   1:  PR[GP1:91,1] = PR[GP1:90,1] + 24.010;
   1:  PR[GP1:91,2] = PR[GP1:90,2] + -39.901;
   1:L PR[91] 10mm/sec CNT100;
   1:  PR[GP1:91,1] = PR[GP1:90,1] + 25.299;
   1:  PR[GP1:91,2] = PR[GP1:90,2] + -39.660;
   1:L PR[91] 10mm/sec CNT100;
   1:  PR[GP1:91,1] = PR[GP1:90,1] + 37.312;
   1:  PR[GP1:91,2] = PR[GP1:90,2] + -34.177;
   1:L PR[91] 10mm/sec CNT100;
   1:  PR[GP1:91,1] = PR[GP1:90,1] + 37.829;
   1:  PR[GP1:91,2] = PR[GP1:90,2] + -33.856;
   1:L PR[91] 10mm/sec CNT100;
   1:  PR[GP1:91,1] = PR[GP1:90,1] + 47.713;
   1:  PR[GP1:91,2] = PR[GP1:90,2] + -24.655;
   1:L PR[91] 10mm/sec CNT100;
   1:  PR[GP1:91,1] = PR[GP1:90,1] + 49.263;
   1:  PR[GP1:91,2] = PR[GP1:90,2] + -21.804;
   1:L PR[91] 10mm/sec CNT100;
   1:  PR[GP1:91,1] = PR[GP1:90,1] + 54.196;
   1:  PR[GP1:91,2] = PR[GP1:90,2] + -12.888;
   1:L PR[91] 10mm/sec CNT100;
   1:  PR[GP1:91,1] = PR[GP1:90,1] + 54.207;
   1:  PR[GP1:91,2] = PR[GP1:90,2] + -12.858;
   1:L PR[91] 10mm/sec CNT100;
   1:  PR[GP1:91,1] = PR[GP1:90,1] + 56.443;
   1:  PR[GP1:91,2] = PR[GP1:90,2] + 0.296;
   1:L PR[91] 10mm/sec CNT100;
   1:  PR[GP1:91,1] = PR[GP1:90,1] + 56.432;
   1:  PR[GP1:91,2] = PR[GP1:90,2] + 0.395;
   1:L PR[91] 10mm/sec CNT100;
   1:  PR[GP1:91,1] = PR[GP1:90,1] + 54.197;
   1:  PR[GP1:91,2] = PR[GP1:90,2] + 13.442;
   1:L PR[91] 10mm/sec CNT100;
   1:  PR[GP1:91,1] = PR[GP1:90,1] + 54.186;
   1:  PR[GP1:91,2] = PR[GP1:90,2] + 13.473;
   1:L PR[91] 10mm/sec CNT100;
   1:  PR[GP1:91,1] = PR[GP1:90,1] + 49.263;
   1:  PR[GP1:91,2] = PR[GP1:90,2] + 22.349;
   1:L PR[91] 10mm/sec CNT100;
   1:  PR[GP1:91,1] = PR[GP1:90,1] + 47.678;
   1:  PR[GP1:91,2] = PR[GP1:90,2] + 25.259;
   1:L PR[91] 10mm/sec CNT100;
   1:  PR[GP1:91,1] = PR[GP1:90,1] + 37.759;
   1:  PR[GP1:91,2] = PR[GP1:90,2] + 34.461;
   1:L PR[91] 10mm/sec CNT100;
   1:  PR[GP1:91,1] = PR[GP1:90,1] + 37.238;
   1:  PR[GP1:91,2] = PR[GP1:90,2] + 34.783;
   1:L PR[91] 10mm/sec CNT100;
   1:  PR[GP1:91,1] = PR[GP1:90,1] + 25.194;
   1:  PR[GP1:91,2] = PR[GP1:90,2] + 40.247;
   1:L PR[91] 10mm/sec CNT100;
   1:  PR[GP1:91,1] = PR[GP1:90,1] + 23.898;
   1:  PR[GP1:91,2] = PR[GP1:90,2] + 40.489;
   1:L PR[91] 10mm/sec CNT100;
   1:  PR[GP1:91,1] = PR[GP1:90,1] + 11.139;
   1:  PR[GP1:91,2] = PR[GP1:90,2] + 41.852;
   1:L PR[91] 10mm/sec CNT100;
   1:  PR[GP1:91,1] = PR[GP1:90,1] + 8.485;
   1:  PR[GP1:91,2] = PR[GP1:90,2] + 41.385;
   1:L PR[91] 10mm/sec CNT100;
   1:  PR[GP1:91,1] = PR[GP1:90,1] + -0.260;
   1:  PR[GP1:91,2] = PR[GP1:90,2] + 39.478;
   1:L PR[91] 10mm/sec CNT100;
   1:  PR[GP1:91,1] = PR[GP1:90,1] + -9.009;
   1:  PR[GP1:91,2] = PR[GP1:90,2] + 41.385;
   1:L PR[91] 10mm/sec CNT100;
   1:  PR[GP1:91,1] = PR[GP1:90,1] + -11.665;
   1:  PR[GP1:91,2] = PR[GP1:90,2] + 41.852;
   1:L PR[91] 10mm/sec CNT100;
   1:  PR[GP1:91,1] = PR[GP1:90,1] + -24.425;
   1:  PR[GP1:91,2] = PR[GP1:90,2] + 40.491;
   1:L PR[91] 10mm/sec CNT100;
   1:  PR[GP1:91,1] = PR[GP1:90,1] + -25.720;
   1:  PR[GP1:91,2] = PR[GP1:90,2] + 40.248;
   1:L PR[91] 10mm/sec CNT100;
   1:  PR[GP1:91,1] = PR[GP1:90,1] + -37.764;
   1:  PR[GP1:91,2] = PR[GP1:90,2] + 34.781;
   1:L PR[91] 10mm/sec CNT100;
   1:  PR[GP1:91,1] = PR[GP1:90,1] + -38.285;
   1:  PR[GP1:91,2] = PR[GP1:90,2] + 34.458;
   1:L PR[91] 10mm/sec CNT100;
   1:  PR[GP1:91,1] = PR[GP1:90,1] + -48.204;
   1:  PR[GP1:91,2] = PR[GP1:90,2] + 25.267;
   1:L PR[91] 10mm/sec CNT100;
   1:  PR[GP1:91,1] = PR[GP1:90,1] + -49.790;
   1:  PR[GP1:91,2] = PR[GP1:90,2] + 22.350;
   1:L PR[91] 10mm/sec CNT100;
   1:  PR[GP1:91,1] = PR[GP1:90,1] + -54.712;
   1:  PR[GP1:91,2] = PR[GP1:90,2] + 13.460;
   1:L PR[91] 10mm/sec CNT100;
   1:  PR[GP1:91,1] = PR[GP1:90,1] + -54.724;
   1:  PR[GP1:91,2] = PR[GP1:90,2] + 13.427;
   1:L PR[91] 10mm/sec CNT100;
   1:  PR[GP1:91,1] = PR[GP1:90,1] + -56.969;
   1:  PR[GP1:91,2] = PR[GP1:90,2] + 0.261;
   1:L PR[91] 10mm/sec CNT100;
   1:  PR[GP1:91,1] = PR[GP1:90,1] + -56.959;
   1:  PR[GP1:91,2] = PR[GP1:90,2] + 0.167;
   1:L PR[91] 10mm/sec CNT100;
   1:  PR[GP1:91,1] = PR[GP1:90,1] + -54.734;
   1:  PR[GP1:91,2] = PR[GP1:90,2] + -12.842;
   1:L PR[91] 10mm/sec CNT100;
   1:  PR[GP1:91,1] = PR[GP1:90,1] + -54.722;
   1:  PR[GP1:91,2] = PR[GP1:90,2] + -12.875;
   1:L PR[91] 10mm/sec CNT100;
   1:  PR[GP1:91,1] = PR[GP1:90,1] + -49.791;
   1:  PR[GP1:91,2] = PR[GP1:90,2] + -21.804;
   1:L PR[91] 10mm/sec CNT100;
   1:  PR[GP1:91,1] = PR[GP1:90,1] + -48.225;
   1:  PR[GP1:91,2] = PR[GP1:90,2] + -24.689;
   1:L PR[91] 10mm/sec CNT100;
   1:  PR[GP1:91,1] = PR[GP1:90,1] + -38.356;
   1:  PR[GP1:91,2] = PR[GP1:90,2] + -33.853;
   1:L PR[91] 10mm/sec CNT100;
   1:  PR[GP1:91,1] = PR[GP1:90,1] + -37.838;
   1:  PR[GP1:91,2] = PR[GP1:90,2] + -34.174;
   1:L PR[91] 10mm/sec CNT100;
   1:  PR[GP1:91,1] = PR[GP1:90,1] + -25.826;
   1:  PR[GP1:91,2] = PR[GP1:90,2] + -39.661;
   1:L PR[91] 10mm/sec CNT100;
   1:  PR[GP1:91,1] = PR[GP1:90,1] + -24.537;
   1:  PR[GP1:91,2] = PR[GP1:90,2] + -39.902;
   1:L PR[91] 10mm/sec CNT100;
   1:  PR[GP1:91,1] = PR[GP1:90,1] + -11.796;
   1:  PR[GP1:91,2] = PR[GP1:90,2] + -41.301;
   1:L PR[91] 10mm/sec CNT100;
   1:  PR[GP1:91,1] = PR[GP1:90,1] + -9.923;
   1:  PR[GP1:91,2] = PR[GP1:90,2] + -40.987;
   1:L PR[91] 10mm/sec CNT100;
   1:  PR[GP1:91,1] = PR[GP1:90,1] + -0.262;
   1:  PR[GP1:91,2] = PR[GP1:90,2] + -38.909;
   1:L PR[91] 10mm/sec CNT100;
   1:  PR[GP1:91,1] = PR[GP1:90,1] + 8.960;
   1:  PR[GP1:91,2] = PR[GP1:90,2] + -41.074;
   1:  PR[GP1:91,3] = PR[GP1:90,3] + 91.805;
   1:L PR[91] 10mm/sec CNT100;
   1:  PR[GP1:91,1] = PR[GP1:90,1] + 11.079;
   1:  PR[GP1:91,2] = PR[GP1:90,2] + -41.430;
   1:L PR[91] 10mm/sec CNT100;
   1:  PR[GP1:91,1] = PR[GP1:90,1] + 23.609;
   1:  PR[GP1:91,2] = PR[GP1:90,2] + -40.053;
   1:L PR[91] 10mm/sec CNT100;
   1:  PR[GP1:91,1] = PR[GP1:90,1] + 25.173;
   1:  PR[GP1:91,2] = PR[GP1:90,2] + -39.761;
   1:L PR[91] 10mm/sec CNT100;
   1:  PR[GP1:91,1] = PR[GP1:90,1] + 36.986;
   1:  PR[GP1:91,2] = PR[GP1:90,2] + -34.368;
   1:L PR[91] 10mm/sec CNT100;
   1:  PR[GP1:91,1] = PR[GP1:90,1] + 37.751;
   1:  PR[GP1:91,2] = PR[GP1:90,2] + -33.894;
   1:L PR[91] 10mm/sec CNT100;
   1:  PR[GP1:91,1] = PR[GP1:90,1] + 47.467;
   1:  PR[GP1:91,2] = PR[GP1:90,2] + -24.863;
   1:L PR[91] 10mm/sec CNT100;
   1:  PR[GP1:91,1] = PR[GP1:90,1] + 47.597;
   1:  PR[GP1:91,2] = PR[GP1:90,2] + -24.706;
   1:L PR[91] 10mm/sec CNT100;
   1:  PR[GP1:91,1] = PR[GP1:90,1] + 54.014;
   1:  PR[GP1:91,2] = PR[GP1:90,2] + -12.903;
   1:L PR[91] 10mm/sec CNT100;
   1:  PR[GP1:91,1] = PR[GP1:90,1] + 56.264;
   1:  PR[GP1:91,2] = PR[GP1:90,2] + 0.291;
   1:L PR[91] 10mm/sec CNT100;
   1:  PR[GP1:91,1] = PR[GP1:90,1] + 54.005;
   1:  PR[GP1:91,2] = PR[GP1:90,2] + 13.485;
   1:L PR[91] 10mm/sec CNT100;
   1:  PR[GP1:91,1] = PR[GP1:90,1] + 47.562;
   1:  PR[GP1:91,2] = PR[GP1:90,2] + 25.309;
   1:L PR[91] 10mm/sec CNT100;
   1:  PR[GP1:91,1] = PR[GP1:90,1] + 47.431;
   1:  PR[GP1:91,2] = PR[GP1:90,2] + 25.467;
   1:L PR[91] 10mm/sec CNT100;
   1:  PR[GP1:91,1] = PR[GP1:90,1] + 37.682;
   1:  PR[GP1:91,2] = PR[GP1:90,2] + 34.498;
   1:L PR[91] 10mm/sec CNT100;
   1:  PR[GP1:91,1] = PR[GP1:90,1] + 36.914;
   1:  PR[GP1:91,2] = PR[GP1:90,2] + 34.974;
   1:L PR[91] 10mm/sec CNT100;
   1:  PR[GP1:91,1] = PR[GP1:90,1] + 25.069;
   1:  PR[GP1:91,2] = PR[GP1:90,2] + 40.347;
   1:L PR[91] 10mm/sec CNT100;
   1:  PR[GP1:91,1] = PR[GP1:90,1] + 23.500;
   1:  PR[GP1:91,2] = PR[GP1:90,2] + 40.641;
   1:L PR[91] 10mm/sec CNT100;
   1:  PR[GP1:91,1] = PR[GP1:90,1] + 10.952;
   1:  PR[GP1:91,2] = PR[GP1:90,2] + 41.981;
   1:L PR[91] 10mm/sec CNT100;
   1:  PR[GP1:91,1] = PR[GP1:90,1] + 7.952;
   1:  PR[GP1:91,2] = PR[GP1:90,2] + 41.453;
   1:L PR[91] 10mm/sec CNT100;
   1:  PR[GP1:91,1] = PR[GP1:90,1] + -0.260;
   1:  PR[GP1:91,2] = PR[GP1:90,2] + 39.662;
   1:L PR[91] 10mm/sec CNT100;
   1:  PR[GP1:91,1] = PR[GP1:90,1] + -8.475;
   1:  PR[GP1:91,2] = PR[GP1:90,2] + 41.453;
   1:L PR[91] 10mm/sec CNT100;
   1:  PR[GP1:91,1] = PR[GP1:90,1] + -11.478;
   1:  PR[GP1:91,2] = PR[GP1:90,2] + 41.980;
   1:L PR[91] 10mm/sec CNT100;
   1:  PR[GP1:91,1] = PR[GP1:90,1] + -24.026;
   1:  PR[GP1:91,2] = PR[GP1:90,2] + 40.642;
   1:L PR[91] 10mm/sec CNT100;
   1:  PR[GP1:91,1] = PR[GP1:90,1] + -25.595;
   1:  PR[GP1:91,2] = PR[GP1:90,2] + 40.348;
   1:L PR[91] 10mm/sec CNT100;
   1:  PR[GP1:91,1] = PR[GP1:90,1] + -37.440;
   1:  PR[GP1:91,2] = PR[GP1:90,2] + 34.971;
   1:L PR[91] 10mm/sec CNT100;
   1:  PR[GP1:91,1] = PR[GP1:90,1] + -38.208;
   1:  PR[GP1:91,2] = PR[GP1:90,2] + 34.496;
   1:L PR[91] 10mm/sec CNT100;
   1:  PR[GP1:91,1] = PR[GP1:90,1] + -47.957;
   1:  PR[GP1:91,2] = PR[GP1:90,2] + 25.475;
   1:L PR[91] 10mm/sec CNT100;
   1:  PR[GP1:91,1] = PR[GP1:90,1] + -48.088;
   1:  PR[GP1:91,2] = PR[GP1:90,2] + 25.317;
   1:L PR[91] 10mm/sec CNT100;
   1:  PR[GP1:91,1] = PR[GP1:90,1] + -54.531;
   1:  PR[GP1:91,2] = PR[GP1:90,2] + 13.474;
   1:L PR[91] 10mm/sec CNT100;
   1:  PR[GP1:91,1] = PR[GP1:90,1] + -56.791;
   1:  PR[GP1:91,2] = PR[GP1:90,2] + 0.267;
   1:L PR[91] 10mm/sec CNT100;
   1:  PR[GP1:91,1] = PR[GP1:90,1] + -54.541;
   1:  PR[GP1:91,2] = PR[GP1:90,2] + -12.886;
   1:L PR[91] 10mm/sec CNT100;
   1:  PR[GP1:91,1] = PR[GP1:90,1] + -48.123;
   1:  PR[GP1:91,2] = PR[GP1:90,2] + -24.714;
   1:L PR[91] 10mm/sec CNT100;
   1:  PR[GP1:91,1] = PR[GP1:90,1] + -47.994;
   1:  PR[GP1:91,2] = PR[GP1:90,2] + -24.870;
   1:L PR[91] 10mm/sec CNT100;
   1:  PR[GP1:91,1] = PR[GP1:90,1] + -38.278;
   1:  PR[GP1:91,2] = PR[GP1:90,2] + -33.892;
   1:L PR[91] 10mm/sec CNT100;
   1:  PR[GP1:91,1] = PR[GP1:90,1] + -37.513;
   1:  PR[GP1:91,2] = PR[GP1:90,2] + -34.365;
   1:L PR[91] 10mm/sec CNT100;
   1:  PR[GP1:91,1] = PR[GP1:90,1] + -25.700;
   1:  PR[GP1:91,2] = PR[GP1:90,2] + -39.762;
   1:L PR[91] 10mm/sec CNT100;
   1:  PR[GP1:91,1] = PR[GP1:90,1] + -24.136;
   1:  PR[GP1:91,2] = PR[GP1:90,2] + -40.054;
   1:L PR[91] 10mm/sec CNT100;
   1:  PR[GP1:91,1] = PR[GP1:90,1] + -11.606;
   1:  PR[GP1:91,2] = PR[GP1:90,2] + -41.429;
   1:L PR[91] 10mm/sec CNT100;
   1:  PR[GP1:91,1] = PR[GP1:90,1] + -9.485;
   1:  PR[GP1:91,2] = PR[GP1:90,2] + -41.074;
   1:L PR[91] 10mm/sec CNT100;
   1:  PR[GP1:91,1] = PR[GP1:90,1] + -0.262;
   1:  PR[GP1:91,2] = PR[GP1:90,2] + -39.090;
   1:L PR[91] 10mm/sec CNT100;
   1:  PR[GP1:91,1] = PR[GP1:90,1] + 8.523;
   1:  PR[GP1:91,2] = PR[GP1:90,2] + -41.161;
   1:  PR[GP1:91,3] = PR[GP1:90,3] + 92.415;
   1:L PR[91] 10mm/sec CNT100;
   1:  PR[GP1:91,1] = PR[GP1:90,1] + 10.890;
   1:  PR[GP1:91,2] = PR[GP1:90,2] + -41.558;
   1:L PR[91] 10mm/sec CNT100;
   1:  PR[GP1:91,1] = PR[GP1:90,1] + 23.209;
   1:  PR[GP1:91,2] = PR[GP1:90,2] + -40.205;
   1:L PR[91] 10mm/sec CNT100;
   1:  PR[GP1:91,1] = PR[GP1:90,1] + 25.047;
   1:  PR[GP1:91,2] = PR[GP1:90,2] + -39.861;
   1:L PR[91] 10mm/sec CNT100;
   1:  PR[GP1:91,1] = PR[GP1:90,1] + 36.661;
   1:  PR[GP1:91,2] = PR[GP1:90,2] + -34.559;
   1:L PR[91] 10mm/sec CNT100;
   1:  PR[GP1:91,1] = PR[GP1:90,1] + 37.673;
   1:  PR[GP1:91,2] = PR[GP1:90,2] + -33.933;
   1:L PR[91] 10mm/sec CNT100;
   1:  PR[GP1:91,1] = PR[GP1:90,1] + 47.225;
   1:  PR[GP1:91,2] = PR[GP1:90,2] + -25.053;
   1:L PR[91] 10mm/sec CNT100;
   1:  PR[GP1:91,1] = PR[GP1:90,1] + 47.499;
   1:  PR[GP1:91,2] = PR[GP1:90,2] + -24.723;
   1:L PR[91] 10mm/sec CNT100;
   1:  PR[GP1:91,1] = PR[GP1:90,1] + 53.845;
   1:  PR[GP1:91,2] = PR[GP1:90,2] + -13.048;
   1:L PR[91] 10mm/sec CNT100;
   1:  PR[GP1:91,1] = PR[GP1:90,1] + 53.896;
   1:  PR[GP1:91,2] = PR[GP1:90,2] + -12.932;
   1:L PR[91] 10mm/sec CNT100;
   1:  PR[GP1:91,1] = PR[GP1:90,1] + 56.107;
   1:  PR[GP1:91,2] = PR[GP1:90,2] + 0.224;
   1:L PR[91] 10mm/sec CNT100;
   1:  PR[GP1:91,2] = PR[GP1:90,2] + 0.232;
   1:L PR[91] 10mm/sec CNT100;
   1:  PR[GP1:91,1] = PR[GP1:90,1] + 54.998;
   1:  PR[GP1:91,2] = PR[GP1:90,2] + 6.763;
   1:L PR[91] 10mm/sec CNT100;
   1:  PR[GP1:91,1] = PR[GP1:90,1] + 53.886;
   1:  PR[GP1:91,2] = PR[GP1:90,2] + 13.518;
   1:L PR[91] 10mm/sec CNT100;
   1:  PR[GP1:91,1] = PR[GP1:90,1] + 53.835;
   1:  PR[GP1:91,2] = PR[GP1:90,2] + 13.633;
   1:L PR[91] 10mm/sec CNT100;
   1:  PR[GP1:91,1] = PR[GP1:90,1] + 47.465;
   1:  PR[GP1:91,2] = PR[GP1:90,2] + 25.325;
   1:L PR[91] 10mm/sec CNT100;
   1:  PR[GP1:91,1] = PR[GP1:90,1] + 47.190;
   1:  PR[GP1:91,2] = PR[GP1:90,2] + 25.657;
   1:L PR[91] 10mm/sec CNT100;
   1:  PR[GP1:91,1] = PR[GP1:90,1] + 37.605;
   1:  PR[GP1:91,2] = PR[GP1:90,2] + 34.536;
   1:L PR[91] 10mm/sec CNT100;
   1:  PR[GP1:91,1] = PR[GP1:90,1] + 36.590;
   1:  PR[GP1:91,2] = PR[GP1:90,2] + 35.164;
   1:L PR[91] 10mm/sec CNT100;
   1:  PR[GP1:91,1] = PR[GP1:90,1] + 24.945;
   1:  PR[GP1:91,2] = PR[GP1:90,2] + 40.447;
   1:L PR[91] 10mm/sec CNT100;
   1:  PR[GP1:91,1] = PR[GP1:90,1] + 23.101;
   1:  PR[GP1:91,2] = PR[GP1:90,2] + 40.792;
   1:L PR[91] 10mm/sec CNT100;
   1:  PR[GP1:91,1] = PR[GP1:90,1] + 10.765;
   1:  PR[GP1:91,2] = PR[GP1:90,2] + 42.109;
   1:L PR[91] 10mm/sec CNT100;
   1:  PR[GP1:91,1] = PR[GP1:90,1] + 7.418;
   1:  PR[GP1:91,2] = PR[GP1:90,2] + 41.521;
   1:L PR[91] 10mm/sec CNT100;
   1:  PR[GP1:91,1] = PR[GP1:90,1] + -0.260;
   1:  PR[GP1:91,2] = PR[GP1:90,2] + 39.846;
   1:L PR[91] 10mm/sec CNT100;
   1:  PR[GP1:91,1] = PR[GP1:90,1] + -7.941;
   1:  PR[GP1:91,2] = PR[GP1:90,2] + 41.520;
   1:L PR[91] 10mm/sec CNT100;
   1:  PR[GP1:91,1] = PR[GP1:90,1] + -11.291;
   1:  PR[GP1:91,2] = PR[GP1:90,2] + 42.109;
   1:L PR[91] 10mm/sec CNT100;
   1:  PR[GP1:91,1] = PR[GP1:90,1] + -23.628;
   1:  PR[GP1:91,2] = PR[GP1:90,2] + 40.793;
   1:L PR[91] 10mm/sec CNT100;
   1:  PR[GP1:91,1] = PR[GP1:90,1] + -25.471;
   1:  PR[GP1:91,2] = PR[GP1:90,2] + 40.448;
   1:L PR[91] 10mm/sec CNT100;
   1:  PR[GP1:91,1] = PR[GP1:90,1] + -37.116;
   1:  PR[GP1:91,2] = PR[GP1:90,2] + 35.162;
   1:L PR[91] 10mm/sec CNT100;
   1:  PR[GP1:91,1] = PR[GP1:90,1] + -38.131;
   1:  PR[GP1:91,2] = PR[GP1:90,2] + 34.533;
   1:L PR[91] 10mm/sec CNT100;
   1:  PR[GP1:91,1] = PR[GP1:90,1] + -47.716;
   1:  PR[GP1:91,2] = PR[GP1:90,2] + 25.664;
   1:L PR[91] 10mm/sec CNT100;
   1:  PR[GP1:91,1] = PR[GP1:90,1] + -47.991;
   1:  PR[GP1:91,2] = PR[GP1:90,2] + 25.333;
   1:L PR[91] 10mm/sec CNT100;
   1:  PR[GP1:91,1] = PR[GP1:90,1] + -54.361;
   1:  PR[GP1:91,2] = PR[GP1:90,2] + 13.620;
   1:L PR[91] 10mm/sec CNT100;
   1:  PR[GP1:91,1] = PR[GP1:90,1] + -54.413;
   1:  PR[GP1:91,2] = PR[GP1:90,2] + 13.503;
   1:L PR[91] 10mm/sec CNT100;
   1:  PR[GP1:91,1] = PR[GP1:90,1] + -56.633;
   1:  PR[GP1:91,2] = PR[GP1:90,2] + 0.334;
   1:L PR[91] 10mm/sec CNT100;
   1:  PR[GP1:91,2] = PR[GP1:90,2] + 0.326;
   1:L PR[91] 10mm/sec CNT100;
   1:  PR[GP1:91,1] = PR[GP1:90,1] + -55.528;
   1:  PR[GP1:91,2] = PR[GP1:90,2] + -6.190;
   1:L PR[91] 10mm/sec CNT100;
   1:  PR[GP1:91,1] = PR[GP1:90,1] + -54.439;
   1:  PR[GP1:91,2] = PR[GP1:90,2] + -12.777;
   1:L PR[91] 10mm/sec CNT100;
   1:  PR[GP1:91,1] = PR[GP1:90,1] + -54.419;
   1:  PR[GP1:91,2] = PR[GP1:90,2] + -12.926;
   1:L PR[91] 10mm/sec CNT100;
   1:  PR[GP1:91,1] = PR[GP1:90,1] + -54.371;
   1:  PR[GP1:91,2] = PR[GP1:90,2] + -13.034;
   1:L PR[91] 10mm/sec CNT100;
   1:  PR[GP1:91,1] = PR[GP1:90,1] + -48.026;
   1:  PR[GP1:91,2] = PR[GP1:90,2] + -24.730;
   1:L PR[91] 10mm/sec CNT100;
   1:  PR[GP1:91,1] = PR[GP1:90,1] + -47.752;
   1:  PR[GP1:91,2] = PR[GP1:90,2] + -25.060;
   1:L PR[91] 10mm/sec CNT100;
   1:  PR[GP1:91,1] = PR[GP1:90,1] + -38.199;
   1:  PR[GP1:91,2] = PR[GP1:90,2] + -33.930;
   1:L PR[91] 10mm/sec CNT100;
   1:  PR[GP1:91,1] = PR[GP1:90,1] + -37.188;
   1:  PR[GP1:91,2] = PR[GP1:90,2] + -34.557;
   1:L PR[91] 10mm/sec CNT100;
   1:  PR[GP1:91,1] = PR[GP1:90,1] + -25.573;
   1:  PR[GP1:91,2] = PR[GP1:90,2] + -39.862;
   1:L PR[91] 10mm/sec CNT100;
   1:  PR[GP1:91,1] = PR[GP1:90,1] + -23.736;
   1:  PR[GP1:91,2] = PR[GP1:90,2] + -40.206;
   1:L PR[91] 10mm/sec CNT100;
   1:  PR[GP1:91,1] = PR[GP1:90,1] + -11.417;
   1:  PR[GP1:91,2] = PR[GP1:90,2] + -41.558;
   1:L PR[91] 10mm/sec CNT100;
   1:  PR[GP1:91,1] = PR[GP1:90,1] + -9.047;
   1:  PR[GP1:91,2] = PR[GP1:90,2] + -41.160;
   1:L PR[91] 10mm/sec CNT100;
   1:  PR[GP1:91,1] = PR[GP1:90,1] + -0.262;
   1:  PR[GP1:91,2] = PR[GP1:90,2] + -39.271;
   1:L PR[91] 10mm/sec CNT100;
   1:  PR[GP1:91,1] = PR[GP1:90,1] + 8.085;
   1:  PR[GP1:91,2] = PR[GP1:90,2] + -41.247;
   1:  PR[GP1:91,3] = PR[GP1:90,3] + 93.025;
   1:L PR[91] 10mm/sec CNT100;
   1:  PR[GP1:91,1] = PR[GP1:90,1] + 10.700;
   1:  PR[GP1:91,2] = PR[GP1:90,2] + -41.687;
   1:L PR[91] 10mm/sec CNT100;
   1:  PR[GP1:91,1] = PR[GP1:90,1] + 22.808;
   1:  PR[GP1:91,2] = PR[GP1:90,2] + -40.356;
   1:L PR[91] 10mm/sec CNT100;
   1:  PR[GP1:91,1] = PR[GP1:90,1] + 24.920;
   1:  PR[GP1:91,2] = PR[GP1:90,2] + -39.962;
   1:L PR[91] 10mm/sec CNT100;
   1:  PR[GP1:91,1] = PR[GP1:90,1] + 36.336;
   1:  PR[GP1:91,2] = PR[GP1:90,2] + -34.751;
   1:L PR[91] 10mm/sec CNT100;
   1:  PR[GP1:91,1] = PR[GP1:90,1] + 37.594;
   1:  PR[GP1:91,2] = PR[GP1:90,2] + -33.971;
   1:L PR[91] 10mm/sec CNT100;
   1:  PR[GP1:91,1] = PR[GP1:90,1] + 46.983;
   1:  PR[GP1:91,2] = PR[GP1:90,2] + -25.243;
   1:L PR[91] 10mm/sec CNT100;
   1:  PR[GP1:91,1] = PR[GP1:90,1] + 47.402;
   1:  PR[GP1:91,2] = PR[GP1:90,2] + -24.739;
   1:L PR[91] 10mm/sec CNT100;
   1:  PR[GP1:91,1] = PR[GP1:90,1] + 53.638;
   1:  PR[GP1:91,2] = PR[GP1:90,2] + -13.265;
   1:L PR[91] 10mm/sec CNT100;
   1:  PR[GP1:91,1] = PR[GP1:90,1] + 53.783;
   1:  PR[GP1:91,2] = PR[GP1:90,2] + -12.937;
   1:L PR[91] 10mm/sec CNT100;
   1:  PR[GP1:91,1] = PR[GP1:90,1] + 55.956;
   1:  PR[GP1:91,2] = PR[GP1:90,2] + -0.005;
   1:L PR[91] 10mm/sec CNT100;
   1:  PR[GP1:91,1] = PR[GP1:90,1] + 55.960;
   1:  PR[GP1:91,2] = PR[GP1:90,2] + 0.234;
   1:L PR[91] 10mm/sec CNT100;
   1:  PR[GP1:91,1] = PR[GP1:90,1] + 53.823;
   1:  PR[GP1:91,2] = PR[GP1:90,2] + 13.152;
   1:L PR[91] 10mm/sec CNT100;
   1:  PR[GP1:91,1] = PR[GP1:90,1] + 53.770;
   1:  PR[GP1:91,2] = PR[GP1:90,2] + 13.530;
   1:L PR[91] 10mm/sec CNT100;
   1:  PR[GP1:91,1] = PR[GP1:90,1] + 53.629;
   1:  PR[GP1:91,2] = PR[GP1:90,2] + 13.849;
   1:L PR[91] 10mm/sec CNT100;
   1:  PR[GP1:91,1] = PR[GP1:90,1] + 47.368;
   1:  PR[GP1:91,2] = PR[GP1:90,2] + 25.341;
   1:L PR[91] 10mm/sec CNT100;
   1:  PR[GP1:91,1] = PR[GP1:90,1] + 46.948;
   1:  PR[GP1:91,2] = PR[GP1:90,2] + 25.846;
   1:L PR[91] 10mm/sec CNT100;
   1:  PR[GP1:91,1] = PR[GP1:90,1] + 37.528;
   1:  PR[GP1:91,2] = PR[GP1:90,2] + 34.573;
   1:L PR[91] 10mm/sec CNT100;
   1:  PR[GP1:91,1] = PR[GP1:90,1] + 36.265;
   1:  PR[GP1:91,2] = PR[GP1:90,2] + 35.355;
   1:L PR[91] 10mm/sec CNT100;
   1:  PR[GP1:91,1] = PR[GP1:90,1] + 24.820;
   1:  PR[GP1:91,2] = PR[GP1:90,2] + 40.547;
   1:L PR[91] 10mm/sec CNT100;
   1:  PR[GP1:91,1] = PR[GP1:90,1] + 22.702;
   1:  PR[GP1:91,2] = PR[GP1:90,2] + 40.943;
   1:L PR[91] 10mm/sec CNT100;
   1:  PR[GP1:91,1] = PR[GP1:90,1] + 10.577;
   1:  PR[GP1:91,2] = PR[GP1:90,2] + 42.238;
   1:L PR[91] 10mm/sec CNT100;
   1:  PR[GP1:91,1] = PR[GP1:90,1] + 6.885;
   1:  PR[GP1:91,2] = PR[GP1:90,2] + 41.588;
   1:L PR[91] 10mm/sec CNT100;
   1:  PR[GP1:91,1] = PR[GP1:90,1] + -0.260;
   1:  PR[GP1:91,2] = PR[GP1:90,2] + 40.030;
   1:L PR[91] 10mm/sec CNT100;
   1:  PR[GP1:91,1] = PR[GP1:90,1] + -7.407;
   1:  PR[GP1:91,2] = PR[GP1:90,2] + 41.588;
   1:L PR[91] 10mm/sec CNT100;
   1:  PR[GP1:91,1] = PR[GP1:90,1] + -11.104;
   1:  PR[GP1:91,2] = PR[GP1:90,2] + 42.237;
   1:L PR[91] 10mm/sec CNT100;
   1:  PR[GP1:91,1] = PR[GP1:90,1] + -23.229;
   1:  PR[GP1:91,2] = PR[GP1:90,2] + 40.944;
   1:L PR[91] 10mm/sec CNT100;
   1:  PR[GP1:91,1] = PR[GP1:90,1] + -25.346;
   1:  PR[GP1:91,2] = PR[GP1:90,2] + 40.548;
   1:L PR[91] 10mm/sec CNT100;
   1:  PR[GP1:91,1] = PR[GP1:90,1] + -36.792;
   1:  PR[GP1:91,2] = PR[GP1:90,2] + 35.352;
   1:L PR[91] 10mm/sec CNT100;
   1:  PR[GP1:91,1] = PR[GP1:90,1] + -38.054;
   1:  PR[GP1:91,2] = PR[GP1:90,2] + 34.571;
   1:L PR[91] 10mm/sec CNT100;
   1:  PR[GP1:91,1] = PR[GP1:90,1] + -47.475;
   1:  PR[GP1:91,2] = PR[GP1:90,2] + 25.854;
   1:L PR[91] 10mm/sec CNT100;
   1:  PR[GP1:91,1] = PR[GP1:90,1] + -47.894;
   1:  PR[GP1:91,2] = PR[GP1:90,2] + 25.349;
   1:L PR[91] 10mm/sec CNT100;
   1:  PR[GP1:91,1] = PR[GP1:90,1] + -54.155;
   1:  PR[GP1:91,2] = PR[GP1:90,2] + 13.836;
   1:L PR[91] 10mm/sec CNT100;
   1:  PR[GP1:91,1] = PR[GP1:90,1] + -54.300;
   1:  PR[GP1:91,2] = PR[GP1:90,2] + 13.508;
   1:L PR[91] 10mm/sec CNT100;
   1:  PR[GP1:91,1] = PR[GP1:90,1] + -56.482;
   1:  PR[GP1:91,2] = PR[GP1:90,2] + 0.565;
   1:L PR[91] 10mm/sec CNT100;
   1:  PR[GP1:91,1] = PR[GP1:90,1] + -56.485;
   1:  PR[GP1:91,2] = PR[GP1:90,2] + 0.316;
   1:L PR[91] 10mm/sec CNT100;
   1:  PR[GP1:91,1] = PR[GP1:90,1] + -54.358;
   1:  PR[GP1:91,2] = PR[GP1:90,2] + -12.554;
   1:L PR[91] 10mm/sec CNT100;
   1:  PR[GP1:91,1] = PR[GP1:90,1] + -54.306;
   1:  PR[GP1:91,2] = PR[GP1:90,2] + -12.931;
   1:L PR[91] 10mm/sec CNT100;
   1:  PR[GP1:91,1] = PR[GP1:90,1] + -54.165;
   1:  PR[GP1:91,2] = PR[GP1:90,2] + -13.251;
   1:L PR[91] 10mm/sec CNT100;
   1:  PR[GP1:91,1] = PR[GP1:90,1] + -47.928;
   1:  PR[GP1:91,2] = PR[GP1:90,2] + -24.747;
   1:L PR[91] 10mm/sec CNT100;
   1:  PR[GP1:91,1] = PR[GP1:90,1] + -47.510;
   1:  PR[GP1:91,2] = PR[GP1:90,2] + -25.251;
   1:L PR[91] 10mm/sec CNT100;
   1:  PR[GP1:91,1] = PR[GP1:90,1] + -38.121;
   1:  PR[GP1:91,2] = PR[GP1:90,2] + -33.968;
   1:L PR[91] 10mm/sec CNT100;
   1:  PR[GP1:91,1] = PR[GP1:90,1] + -36.862;
   1:  PR[GP1:91,2] = PR[GP1:90,2] + -34.748;
   1:L PR[91] 10mm/sec CNT100;
   1:  PR[GP1:91,1] = PR[GP1:90,1] + -25.447;
   1:  PR[GP1:91,2] = PR[GP1:90,2] + -39.962;
   1:L PR[91] 10mm/sec CNT100;
   1:  PR[GP1:91,1] = PR[GP1:90,1] + -23.336;
   1:  PR[GP1:91,2] = PR[GP1:90,2] + -40.357;
   1:L PR[91] 10mm/sec CNT100;
   1:  PR[GP1:91,1] = PR[GP1:90,1] + -11.228;
   1:  PR[GP1:91,2] = PR[GP1:90,2] + -41.686;
   1:L PR[91] 10mm/sec CNT100;
   1:  PR[GP1:91,1] = PR[GP1:90,1] + -8.609;
   1:  PR[GP1:91,2] = PR[GP1:90,2] + -41.247;
   1:L PR[91] 10mm/sec CNT100;
   1:  PR[GP1:91,1] = PR[GP1:90,1] + -0.262;
   1:  PR[GP1:91,2] = PR[GP1:90,2] + -39.452;
   1:L PR[91] 10mm/sec CNT100;
   1:  PR[GP1:91,1] = PR[GP1:90,1] + 7.647;
   1:  PR[GP1:91,2] = PR[GP1:90,2] + -41.334;
   1:  PR[GP1:91,3] = PR[GP1:90,3] + 93.635;
   1:L PR[91] 10mm/sec CNT100;
   1:  PR[GP1:91,1] = PR[GP1:90,1] + 10.511;
   1:  PR[GP1:91,2] = PR[GP1:90,2] + -41.815;
   1:L PR[91] 10mm/sec CNT100;
   1:  PR[GP1:91,1] = PR[GP1:90,1] + 22.408;
   1:  PR[GP1:91,2] = PR[GP1:90,2] + -40.508;
   1:L PR[91] 10mm/sec CNT100;
   1:  PR[GP1:91,1] = PR[GP1:90,1] + 24.794;
   1:  PR[GP1:91,2] = PR[GP1:90,2] + -40.062;
   1:L PR[91] 10mm/sec CNT100;
   1:  PR[GP1:91,1] = PR[GP1:90,1] + 36.010;
   1:  PR[GP1:91,2] = PR[GP1:90,2] + -34.942;
   1:L PR[91] 10mm/sec CNT100;
   1:  PR[GP1:91,1] = PR[GP1:90,1] + 37.516;
   1:  PR[GP1:91,2] = PR[GP1:90,2] + -34.009;
   1:L PR[91] 10mm/sec CNT100;
   1:  PR[GP1:91,1] = PR[GP1:90,1] + 46.741;
   1:  PR[GP1:91,2] = PR[GP1:90,2] + -25.434;
   1:L PR[91] 10mm/sec CNT100;
   1:  PR[GP1:91,1] = PR[GP1:90,1] + 47.304;
   1:  PR[GP1:91,2] = PR[GP1:90,2] + -24.756;
   1:L PR[91] 10mm/sec CNT100;
   1:  PR[GP1:91,1] = PR[GP1:90,1] + 53.432;
   1:  PR[GP1:91,2] = PR[GP1:90,2] + -13.481;
   1:L PR[91] 10mm/sec CNT100;
   1:  PR[GP1:91,1] = PR[GP1:90,1] + 53.670;
   1:  PR[GP1:91,2] = PR[GP1:90,2] + -12.943;
   1:L PR[91] 10mm/sec CNT100;
   1:  PR[GP1:91,1] = PR[GP1:90,1] + 55.805;
   1:  PR[GP1:91,2] = PR[GP1:90,2] + -0.237;
   1:L PR[91] 10mm/sec CNT100;
   1:  PR[GP1:91,1] = PR[GP1:90,1] + 55.809;
   1:  PR[GP1:91,2] = PR[GP1:90,2] + 0.075;
   1:L PR[91] 10mm/sec CNT100;
   1:  PR[GP1:91,1] = PR[GP1:90,1] + 55.836;
   1:  PR[GP1:91,2] = PR[GP1:90,2] + 0.271;
   1:L PR[91] 10mm/sec CNT100;
   1:  PR[GP1:91,1] = PR[GP1:90,1] + 53.742;
   1:  PR[GP1:91,2] = PR[GP1:90,2] + 12.928;
   1:L PR[91] 10mm/sec CNT100;
   1:  PR[GP1:91,1] = PR[GP1:90,1] + 53.657;
   1:  PR[GP1:91,2] = PR[GP1:90,2] + 13.534;
   1:L PR[91] 10mm/sec CNT100;
   1:  PR[GP1:91,1] = PR[GP1:90,1] + 53.423;
   1:  PR[GP1:91,2] = PR[GP1:90,2] + 14.065;
   1:L PR[91] 10mm/sec CNT100;
   1:  PR[GP1:91,1] = PR[GP1:90,1] + 47.271;
   1:  PR[GP1:91,2] = PR[GP1:90,2] + 25.357;
   1:L PR[91] 10mm/sec CNT100;
   1:  PR[GP1:91,1] = PR[GP1:90,1] + 46.707;
   1:  PR[GP1:91,2] = PR[GP1:90,2] + 26.036;
   1:L PR[91] 10mm/sec CNT100;
   1:  PR[GP1:91,1] = PR[GP1:90,1] + 37.450;
   1:  PR[GP1:91,2] = PR[GP1:90,2] + 34.611;
   1:L PR[91] 10mm/sec CNT100;
   1:  PR[GP1:91,1] = PR[GP1:90,1] + 35.941;
   1:  PR[GP1:91,2] = PR[GP1:90,2] + 35.545;
   1:L PR[91] 10mm/sec CNT100;
   1:  PR[GP1:91,1] = PR[GP1:90,1] + 24.696;
   1:  PR[GP1:91,2] = PR[GP1:90,2] + 40.647;
   1:L PR[91] 10mm/sec CNT100;
   1:  PR[GP1:91,1] = PR[GP1:90,1] + 22.304;
   1:  PR[GP1:91,2] = PR[GP1:90,2] + 41.094;
   1:L PR[91] 10mm/sec CNT100;
   1:  PR[GP1:91,1] = PR[GP1:90,1] + 10.390;
   1:  PR[GP1:91,2] = PR[GP1:90,2] + 42.366;
   1:L PR[91] 10mm/sec CNT100;
   1:  PR[GP1:91,1] = PR[GP1:90,1] + 6.351;
   1:  PR[GP1:91,2] = PR[GP1:90,2] + 41.656;
   1:L PR[91] 10mm/sec CNT100;
   1:  PR[GP1:91,1] = PR[GP1:90,1] + -0.260;
   1:  PR[GP1:91,2] = PR[GP1:90,2] + 40.214;
   1:L PR[91] 10mm/sec CNT100;
   1:  PR[GP1:91,1] = PR[GP1:90,1] + -6.874;
   1:  PR[GP1:91,2] = PR[GP1:90,2] + 41.656;
   1:L PR[91] 10mm/sec CNT100;
   1:  PR[GP1:91,1] = PR[GP1:90,1] + -10.917;
   1:  PR[GP1:91,2] = PR[GP1:90,2] + 42.366;
   1:L PR[91] 10mm/sec CNT100;
   1:  PR[GP1:91,1] = PR[GP1:90,1] + -22.831;
   1:  PR[GP1:91,2] = PR[GP1:90,2] + 41.095;
   1:L PR[91] 10mm/sec CNT100;
   1:  PR[GP1:91,1] = PR[GP1:90,1] + -25.222;
   1:  PR[GP1:91,2] = PR[GP1:90,2] + 40.648;
   1:L PR[91] 10mm/sec CNT100;
   1:  PR[GP1:91,1] = PR[GP1:90,1] + -36.468;
   1:  PR[GP1:91,2] = PR[GP1:90,2] + 35.543;
   1:L PR[91] 10mm/sec CNT100;
   1:  PR[GP1:91,1] = PR[GP1:90,1] + -37.976;
   1:  PR[GP1:91,2] = PR[GP1:90,2] + 34.608;
   1:L PR[91] 10mm/sec CNT100;
   1:  PR[GP1:91,1] = PR[GP1:90,1] + -47.233;
   1:  PR[GP1:91,2] = PR[GP1:90,2] + 26.043;
   1:L PR[91] 10mm/sec CNT100;
   1:  PR[GP1:91,1] = PR[GP1:90,1] + -47.797;
   1:  PR[GP1:91,2] = PR[GP1:90,2] + 25.365;
   1:L PR[91] 10mm/sec CNT100;
   1:  PR[GP1:91,1] = PR[GP1:90,1] + -53.949;
   1:  PR[GP1:91,2] = PR[GP1:90,2] + 14.052;
   1:L PR[91] 10mm/sec CNT100;
   1:  PR[GP1:91,1] = PR[GP1:90,1] + -54.187;
   1:  PR[GP1:91,2] = PR[GP1:90,2] + 13.513;
   1:L PR[91] 10mm/sec CNT100;
   1:  PR[GP1:91,1] = PR[GP1:90,1] + -56.331;
   1:  PR[GP1:91,2] = PR[GP1:90,2] + 0.795;
   1:L PR[91] 10mm/sec CNT100;
   1:  PR[GP1:91,1] = PR[GP1:90,1] + -56.335;
   1:  PR[GP1:91,2] = PR[GP1:90,2] + 0.483;
   1:L PR[91] 10mm/sec CNT100;
   1:  PR[GP1:91,1] = PR[GP1:90,1] + -56.362;
   1:  PR[GP1:91,2] = PR[GP1:90,2] + 0.287;
   1:L PR[91] 10mm/sec CNT100;
   1:  PR[GP1:91,1] = PR[GP1:90,1] + -54.277;
   1:  PR[GP1:91,2] = PR[GP1:90,2] + -12.330;
   1:L PR[91] 10mm/sec CNT100;
   1:  PR[GP1:91,1] = PR[GP1:90,1] + -54.193;
   1:  PR[GP1:91,2] = PR[GP1:90,2] + -12.937;
   1:L PR[91] 10mm/sec CNT100;
   1:  PR[GP1:91,1] = PR[GP1:90,1] + -53.958;
   1:  PR[GP1:91,2] = PR[GP1:90,2] + -13.468;
   1:L PR[91] 10mm/sec CNT100;
   1:  PR[GP1:91,1] = PR[GP1:90,1] + -47.830;
   1:  PR[GP1:91,2] = PR[GP1:90,2] + -24.763;
   1:L PR[91] 10mm/sec CNT100;
   1:  PR[GP1:91,1] = PR[GP1:90,1] + -47.268;
   1:  PR[GP1:91,2] = PR[GP1:90,2] + -25.441;
   1:L PR[91] 10mm/sec CNT100;
   1:  PR[GP1:91,1] = PR[GP1:90,1] + -38.043;
   1:  PR[GP1:91,2] = PR[GP1:90,2] + -34.007;
   1:L PR[91] 10mm/sec CNT100;
   1:  PR[GP1:91,1] = PR[GP1:90,1] + -36.537;
   1:  PR[GP1:91,2] = PR[GP1:90,2] + -34.939;
   1:L PR[91] 10mm/sec CNT100;
   1:  PR[GP1:91,1] = PR[GP1:90,1] + -25.321;
   1:  PR[GP1:91,2] = PR[GP1:90,2] + -40.063;
   1:L PR[91] 10mm/sec CNT100;
   1:  PR[GP1:91,1] = PR[GP1:90,1] + -22.935;
   1:  PR[GP1:91,2] = PR[GP1:90,2] + -40.509;
   1:L PR[91] 10mm/sec CNT100;
   1:  PR[GP1:91,1] = PR[GP1:90,1] + -11.039;
   1:  PR[GP1:91,2] = PR[GP1:90,2] + -41.815;
   1:L PR[91] 10mm/sec CNT100;
   1:  PR[GP1:91,1] = PR[GP1:90,1] + -8.171;
   1:  PR[GP1:91,2] = PR[GP1:90,2] + -41.334;
   1:L PR[91] 10mm/sec CNT100;
   1:  PR[GP1:91,1] = PR[GP1:90,1] + -0.262;
   1:  PR[GP1:91,2] = PR[GP1:90,2] + -39.633;
   1:L PR[91] 10mm/sec CNT100;
   1:  PR[GP1:91,1] = PR[GP1:90,1] + 7.209;
   1:  PR[GP1:91,2] = PR[GP1:90,2] + -41.421;
   1:  PR[GP1:91,3] = PR[GP1:90,3] + 94.245;
   1:L PR[91] 10mm/sec CNT100;
   1:  PR[GP1:91,1] = PR[GP1:90,1] + 10.322;
   1:  PR[GP1:91,2] = PR[GP1:90,2] + -41.943;
   1:L PR[91] 10mm/sec CNT100;
   1:  PR[GP1:91,1] = PR[GP1:90,1] + 22.007;
   1:  PR[GP1:91,2] = PR[GP1:90,2] + -40.660;
   1:L PR[91] 10mm/sec CNT100;
   1:  PR[GP1:91,1] = PR[GP1:90,1] + 24.668;
   1:  PR[GP1:91,2] = PR[GP1:90,2] + -40.162;
   1:L PR[91] 10mm/sec CNT100;
   1:  PR[GP1:91,1] = PR[GP1:90,1] + 35.685;
   1:  PR[GP1:91,2] = PR[GP1:90,2] + -35.133;
   1:L PR[91] 10mm/sec CNT100;
   1:  PR[GP1:91,1] = PR[GP1:90,1] + 37.438;
   1:  PR[GP1:91,2] = PR[GP1:90,2] + -34.048;
   1:L PR[91] 10mm/sec CNT100;
   1:  PR[GP1:91,1] = PR[GP1:90,1] + 46.499;
   1:  PR[GP1:91,2] = PR[GP1:90,2] + -25.624;
   1:L PR[91] 10mm/sec CNT100;
   1:  PR[GP1:91,1] = PR[GP1:90,1] + 47.206;
   1:  PR[GP1:91,2] = PR[GP1:90,2] + -24.773;
   1:L PR[91] 10mm/sec CNT100;
   1:  PR[GP1:91,1] = PR[GP1:90,1] + 53.226;
   1:  PR[GP1:91,2] = PR[GP1:90,2] + -13.697;
   1:L PR[91] 10mm/sec CNT100;
   1:  PR[GP1:91,1] = PR[GP1:90,1] + 53.557;
   1:  PR[GP1:91,2] = PR[GP1:90,2] + -12.948;
   1:L PR[91] 10mm/sec CNT100;
   1:  PR[GP1:91,1] = PR[GP1:90,1] + 55.654;
   1:  PR[GP1:91,2] = PR[GP1:90,2] + -0.468;
   1:L PR[91] 10mm/sec CNT100;
   1:  PR[GP1:91,1] = PR[GP1:90,1] + 55.658;
   1:  PR[GP1:91,2] = PR[GP1:90,2] + -0.161;
   1:L PR[91] 10mm/sec CNT100;
   1:  PR[GP1:91,1] = PR[GP1:90,1] + 55.718;
   1:  PR[GP1:91,2] = PR[GP1:90,2] + 0.271;
   1:L PR[91] 10mm/sec CNT100;
   1:  PR[GP1:91,1] = PR[GP1:90,1] + 53.661;
   1:  PR[GP1:91,2] = PR[GP1:90,2] + 12.703;
   1:L PR[91] 10mm/sec CNT100;
   1:  PR[GP1:91,1] = PR[GP1:90,1] + 53.544;
   1:  PR[GP1:91,2] = PR[GP1:90,2] + 13.539;
   1:L PR[91] 10mm/sec CNT100;
   1:  PR[GP1:91,1] = PR[GP1:90,1] + 53.217;
   1:  PR[GP1:91,2] = PR[GP1:90,2] + 14.281;
   1:L PR[91] 10mm/sec CNT100;
   1:  PR[GP1:91,1] = PR[GP1:90,1] + 47.173;
   1:  PR[GP1:91,2] = PR[GP1:90,2] + 25.373;
   1:L PR[91] 10mm/sec CNT100;
   1:  PR[GP1:91,1] = PR[GP1:90,1] + 46.466;
   1:  PR[GP1:91,2] = PR[GP1:90,2] + 26.225;
   1:L PR[91] 10mm/sec CNT100;
   1:  PR[GP1:91,1] = PR[GP1:90,1] + 37.373;
   1:  PR[GP1:91,2] = PR[GP1:90,2] + 34.648;
   1:L PR[91] 10mm/sec CNT100;
   1:  PR[GP1:91,1] = PR[GP1:90,1] + 35.617;
   1:  PR[GP1:91,2] = PR[GP1:90,2] + 35.736;
   1:L PR[91] 10mm/sec CNT100;
   1:  PR[GP1:91,1] = PR[GP1:90,1] + 24.571;
   1:  PR[GP1:91,2] = PR[GP1:90,2] + 40.747;
   1:L PR[91] 10mm/sec CNT100;
   1:  PR[GP1:91,1] = PR[GP1:90,1] + 21.905;
   1:  PR[GP1:91,2] = PR[GP1:90,2] + 41.245;
   1:L PR[91] 10mm/sec CNT100;
   1:  PR[GP1:91,1] = PR[GP1:90,1] + 10.203;
   1:  PR[GP1:91,2] = PR[GP1:90,2] + 42.495;
   1:L PR[91] 10mm/sec CNT100;
   1:  PR[GP1:91,1] = PR[GP1:90,1] + 5.818;
   1:  PR[GP1:91,2] = PR[GP1:90,2] + 41.724;
   1:L PR[91] 10mm/sec CNT100;
   1:  PR[GP1:91,1] = PR[GP1:90,1] + -0.260;
   1:  PR[GP1:91,2] = PR[GP1:90,2] + 40.398;
   1:L PR[91] 10mm/sec CNT100;
   1:  PR[GP1:91,1] = PR[GP1:90,1] + -6.340;
   1:  PR[GP1:91,2] = PR[GP1:90,2] + 41.723;
   1:L PR[91] 10mm/sec CNT100;
   1:  PR[GP1:91,1] = PR[GP1:90,1] + -10.730;
   1:  PR[GP1:91,2] = PR[GP1:90,2] + 42.494;
   1:L PR[91] 10mm/sec CNT100;
   1:  PR[GP1:91,1] = PR[GP1:90,1] + -22.432;
   1:  PR[GP1:91,2] = PR[GP1:90,2] + 41.246;
   1:L PR[91] 10mm/sec CNT100;
   1:  PR[GP1:91,1] = PR[GP1:90,1] + -25.097;
   1:  PR[GP1:91,2] = PR[GP1:90,2] + 40.748;
   1:L PR[91] 10mm/sec CNT100;
   1:  PR[GP1:91,1] = PR[GP1:90,1] + -36.143;
   1:  PR[GP1:91,2] = PR[GP1:90,2] + 35.733;
   1:L PR[91] 10mm/sec CNT100;
   1:  PR[GP1:91,1] = PR[GP1:90,1] + -37.899;
   1:  PR[GP1:91,2] = PR[GP1:90,2] + 34.646;
   1:L PR[91] 10mm/sec CNT100;
   1:  PR[GP1:91,1] = PR[GP1:90,1] + -46.992;
   1:  PR[GP1:91,2] = PR[GP1:90,2] + 26.233;
   1:L PR[91] 10mm/sec CNT100;
   1:  PR[GP1:91,1] = PR[GP1:90,1] + -47.700;
   1:  PR[GP1:91,2] = PR[GP1:90,2] + 25.380;
   1:L PR[91] 10mm/sec CNT100;
   1:  PR[GP1:91,1] = PR[GP1:90,1] + -53.743;
   1:  PR[GP1:91,2] = PR[GP1:90,2] + 14.268;
   1:L PR[91] 10mm/sec CNT100;
   1:  PR[GP1:91,1] = PR[GP1:90,1] + -54.074;
   1:  PR[GP1:91,2] = PR[GP1:90,2] + 13.518;
   1:L PR[91] 10mm/sec CNT100;
   1:  PR[GP1:91,1] = PR[GP1:90,1] + -56.181;
   1:  PR[GP1:91,2] = PR[GP1:90,2] + 1.026;
   1:L PR[91] 10mm/sec CNT100;
   1:  PR[GP1:91,1] = PR[GP1:90,1] + -56.184;
   1:  PR[GP1:91,2] = PR[GP1:90,2] + 0.719;
   1:L PR[91] 10mm/sec CNT100;
   1:  PR[GP1:91,1] = PR[GP1:90,1] + -56.244;
   1:  PR[GP1:91,2] = PR[GP1:90,2] + 0.287;
   1:L PR[91] 10mm/sec CNT100;
   1:  PR[GP1:91,1] = PR[GP1:90,1] + -54.196;
   1:  PR[GP1:91,2] = PR[GP1:90,2] + -12.107;
   1:L PR[91] 10mm/sec CNT100;
   1:  PR[GP1:91,1] = PR[GP1:90,1] + -54.080;
   1:  PR[GP1:91,2] = PR[GP1:90,2] + -12.942;
   1:L PR[91] 10mm/sec CNT100;
   1:  PR[GP1:91,1] = PR[GP1:90,1] + -53.752;
   1:  PR[GP1:91,2] = PR[GP1:90,2] + -13.684;
   1:L PR[91] 10mm/sec CNT100;
   1:  PR[GP1:91,1] = PR[GP1:90,1] + -47.733;
   1:  PR[GP1:91,2] = PR[GP1:90,2] + -24.780;
   1:L PR[91] 10mm/sec CNT100;
   1:  PR[GP1:91,1] = PR[GP1:90,1] + -47.026;
   1:  PR[GP1:91,2] = PR[GP1:90,2] + -25.631;
   1:L PR[91] 10mm/sec CNT100;
   1:  PR[GP1:91,1] = PR[GP1:90,1] + -37.964;
   1:  PR[GP1:91,2] = PR[GP1:90,2] + -34.045;
   1:L PR[91] 10mm/sec CNT100;
   1:  PR[GP1:91,1] = PR[GP1:90,1] + -36.212;
   1:  PR[GP1:91,2] = PR[GP1:90,2] + -35.130;
   1:L PR[91] 10mm/sec CNT100;
   1:  PR[GP1:91,1] = PR[GP1:90,1] + -25.195;
   1:  PR[GP1:91,2] = PR[GP1:90,2] + -40.163;
   1:L PR[91] 10mm/sec CNT100;
   1:  PR[GP1:91,1] = PR[GP1:90,1] + -22.535;
   1:  PR[GP1:91,2] = PR[GP1:90,2] + -40.661;
   1:L PR[91] 10mm/sec CNT100;
   1:  PR[GP1:91,1] = PR[GP1:90,1] + -10.850;
   1:  PR[GP1:91,2] = PR[GP1:90,2] + -41.943;
   1:L PR[91] 10mm/sec CNT100;
   1:  PR[GP1:91,1] = PR[GP1:90,1] + -7.733;
   1:  PR[GP1:91,2] = PR[GP1:90,2] + -41.421;
   1:L PR[91] 10mm/sec CNT100;
   1:  PR[GP1:91,1] = PR[GP1:90,1] + -0.262;
   1:  PR[GP1:91,2] = PR[GP1:90,2] + -39.814;
   1:L PR[91] 10mm/sec CNT100;
   1:  PR[GP1:91,1] = PR[GP1:90,1] + 6.771;
   1:  PR[GP1:91,2] = PR[GP1:90,2] + -41.508;
   1:  PR[GP1:91,3] = PR[GP1:90,3] + 94.855;
   1:L PR[91] 10mm/sec CNT100;
   1:  PR[GP1:91,1] = PR[GP1:90,1] + 10.132;
   1:  PR[GP1:91,2] = PR[GP1:90,2] + -42.072;
   1:L PR[91] 10mm/sec CNT100;
   1:  PR[GP1:91,1] = PR[GP1:90,1] + 21.607;
   1:  PR[GP1:91,2] = PR[GP1:90,2] + -40.811;
   1:L PR[91] 10mm/sec CNT100;
   1:  PR[GP1:91,1] = PR[GP1:90,1] + 24.542;
   1:  PR[GP1:91,2] = PR[GP1:90,2] + -40.263;
   1:L PR[91] 10mm/sec CNT100;
   1:  PR[GP1:91,1] = PR[GP1:90,1] + 35.360;
   1:  PR[GP1:91,2] = PR[GP1:90,2] + -35.324;
   1:L PR[91] 10mm/sec CNT100;
   1:  PR[GP1:91,1] = PR[GP1:90,1] + 37.359;
   1:  PR[GP1:91,2] = PR[GP1:90,2] + -34.086;
   1:L PR[91] 10mm/sec CNT100;
   1:  PR[GP1:91,1] = PR[GP1:90,1] + 46.258;
   1:  PR[GP1:91,2] = PR[GP1:90,2] + -25.814;
   1:L PR[91] 10mm/sec CNT100;
   1:  PR[GP1:91,1] = PR[GP1:90,1] + 47.109;
   1:  PR[GP1:91,2] = PR[GP1:90,2] + -24.789;
   1:L PR[91] 10mm/sec CNT100;
   1:  PR[GP1:91,1] = PR[GP1:90,1] + 53.020;
   1:  PR[GP1:91,2] = PR[GP1:90,2] + -13.913;
   1:L PR[91] 10mm/sec CNT100;
   1:  PR[GP1:91,1] = PR[GP1:90,1] + 53.444;
   1:  PR[GP1:91,2] = PR[GP1:90,2] + -12.953;
   1:L PR[91] 10mm/sec CNT100;
   1:  PR[GP1:91,1] = PR[GP1:90,1] + 55.503;
   1:  PR[GP1:91,2] = PR[GP1:90,2] + -0.699;
   1:L PR[91] 10mm/sec CNT100;
   1:  PR[GP1:91,1] = PR[GP1:90,1] + 55.507;
   1:  PR[GP1:91,2] = PR[GP1:90,2] + -0.397;
   1:L PR[91] 10mm/sec CNT100;
   1:  PR[GP1:91,1] = PR[GP1:90,1] + 55.600;
   1:  PR[GP1:91,2] = PR[GP1:90,2] + 0.271;
   1:L PR[91] 10mm/sec CNT100;
   1:  PR[GP1:91,1] = PR[GP1:90,1] + 53.580;
   1:  PR[GP1:91,2] = PR[GP1:90,2] + 12.479;
   1:L PR[91] 10mm/sec CNT100;
   1:  PR[GP1:91,1] = PR[GP1:90,1] + 53.432;
   1:  PR[GP1:91,2] = PR[GP1:90,2] + 13.543;
   1:L PR[91] 10mm/sec CNT100;
   1:  PR[GP1:91,1] = PR[GP1:90,1] + 53.011;
   1:  PR[GP1:91,2] = PR[GP1:90,2] + 14.497;
   1:L PR[91] 10mm/sec CNT100;
   1:  PR[GP1:91,1] = PR[GP1:90,1] + 47.076;
   1:  PR[GP1:91,2] = PR[GP1:90,2] + 25.389;
   1:L PR[91] 10mm/sec CNT100;
   1:  PR[GP1:91,1] = PR[GP1:90,1] + 46.225;
   1:  PR[GP1:91,2] = PR[GP1:90,2] + 26.415;
   1:L PR[91] 10mm/sec CNT100;
   1:  PR[GP1:91,1] = PR[GP1:90,1] + 37.296;
   1:  PR[GP1:91,2] = PR[GP1:90,2] + 34.686;
   1:L PR[91] 10mm/sec CNT100;
   1:  PR[GP1:91,1] = PR[GP1:90,1] + 35.293;
   1:  PR[GP1:91,2] = PR[GP1:90,2] + 35.926;
   1:L PR[91] 10mm/sec CNT100;
   1:  PR[GP1:91,1] = PR[GP1:90,1] + 24.447;
   1:  PR[GP1:91,2] = PR[GP1:90,2] + 40.847;
   1:L PR[91] 10mm/sec CNT100;
   1:  PR[GP1:91,1] = PR[GP1:90,1] + 21.506;
   1:  PR[GP1:91,2] = PR[GP1:90,2] + 41.396;
   1:L PR[91] 10mm/sec CNT100;
   1:  PR[GP1:91,1] = PR[GP1:90,1] + 10.016;
   1:  PR[GP1:91,2] = PR[GP1:90,2] + 42.623;
   1:L PR[91] 10mm/sec CNT100;
   1:  PR[GP1:91,1] = PR[GP1:90,1] + 5.284;
   1:  PR[GP1:91,2] = PR[GP1:90,2] + 41.791;
   1:L PR[91] 10mm/sec CNT100;
   1:  PR[GP1:91,1] = PR[GP1:90,1] + -0.260;
   1:  PR[GP1:91,2] = PR[GP1:90,2] + 40.582;
   1:L PR[91] 10mm/sec CNT100;
   1:  PR[GP1:91,1] = PR[GP1:90,1] + -5.806;
   1:  PR[GP1:91,2] = PR[GP1:90,2] + 41.791;
   1:L PR[91] 10mm/sec CNT100;
   1:  PR[GP1:91,1] = PR[GP1:90,1] + -10.543;
   1:  PR[GP1:91,2] = PR[GP1:90,2] + 42.623;
   1:L PR[91] 10mm/sec CNT100;
   1:  PR[GP1:91,1] = PR[GP1:90,1] + -22.034;
   1:  PR[GP1:91,2] = PR[GP1:90,2] + 41.397;
   1:L PR[91] 10mm/sec CNT100;
   1:  PR[GP1:91,1] = PR[GP1:90,1] + -24.973;
   1:  PR[GP1:91,2] = PR[GP1:90,2] + 40.848;
   1:L PR[91] 10mm/sec CNT100;
   1:  PR[GP1:91,1] = PR[GP1:90,1] + -35.819;
   1:  PR[GP1:91,2] = PR[GP1:90,2] + 35.924;
   1:L PR[91] 10mm/sec CNT100;
   1:  PR[GP1:91,1] = PR[GP1:90,1] + -37.822;
   1:  PR[GP1:91,2] = PR[GP1:90,2] + 34.684;
   1:L PR[91] 10mm/sec CNT100;
   1:  PR[GP1:91,1] = PR[GP1:90,1] + -46.751;
   1:  PR[GP1:91,2] = PR[GP1:90,2] + 26.422;
   1:L PR[91] 10mm/sec CNT100;
   1:  PR[GP1:91,1] = PR[GP1:90,1] + -47.602;
   1:  PR[GP1:91,2] = PR[GP1:90,2] + 25.396;
   1:L PR[91] 10mm/sec CNT100;
   1:  PR[GP1:91,1] = PR[GP1:90,1] + -53.537;
   1:  PR[GP1:91,2] = PR[GP1:90,2] + 14.484;
   1:L PR[91] 10mm/sec CNT100;
   1:  PR[GP1:91,1] = PR[GP1:90,1] + -53.961;
   1:  PR[GP1:91,2] = PR[GP1:90,2] + 13.523;
   1:L PR[91] 10mm/sec CNT100;
   1:  PR[GP1:91,1] = PR[GP1:90,1] + -56.030;
   1:  PR[GP1:91,2] = PR[GP1:90,2] + 1.257;
   1:L PR[91] 10mm/sec CNT100;
   1:  PR[GP1:91,1] = PR[GP1:90,1] + -56.033;
   1:  PR[GP1:91,2] = PR[GP1:90,2] + 0.955;
   1:L PR[91] 10mm/sec CNT100;
   1:  PR[GP1:91,1] = PR[GP1:90,1] + -56.126;
   1:  PR[GP1:91,2] = PR[GP1:90,2] + 0.287;
   1:L PR[91] 10mm/sec CNT100;
   1:  PR[GP1:91,1] = PR[GP1:90,1] + -54.115;
   1:  PR[GP1:91,2] = PR[GP1:90,2] + -11.883;
   1:L PR[91] 10mm/sec CNT100;
   1:  PR[GP1:91,1] = PR[GP1:90,1] + -53.967;
   1:  PR[GP1:91,2] = PR[GP1:90,2] + -12.947;
   1:L PR[91] 10mm/sec CNT100;
   1:  PR[GP1:91,1] = PR[GP1:90,1] + -53.546;
   1:  PR[GP1:91,2] = PR[GP1:90,2] + -13.901;
   1:L PR[91] 10mm/sec CNT100;
   1:  PR[GP1:91,1] = PR[GP1:90,1] + -47.635;
   1:  PR[GP1:91,2] = PR[GP1:90,2] + -24.796;
   1:L PR[91] 10mm/sec CNT100;
   1:  PR[GP1:91,1] = PR[GP1:90,1] + -46.784;
   1:  PR[GP1:91,2] = PR[GP1:90,2] + -25.821;
   1:L PR[91] 10mm/sec CNT100;
   1:  PR[GP1:91,1] = PR[GP1:90,1] + -37.886;
   1:  PR[GP1:91,2] = PR[GP1:90,2] + -34.083;
   1:L PR[91] 10mm/sec CNT100;
   1:  PR[GP1:91,1] = PR[GP1:90,1] + -35.886;
   1:  PR[GP1:91,2] = PR[GP1:90,2] + -35.322;
   1:L PR[91] 10mm/sec CNT100;
   1:  PR[GP1:91,1] = PR[GP1:90,1] + -25.069;
   1:  PR[GP1:91,2] = PR[GP1:90,2] + -40.263;
   1:L PR[91] 10mm/sec CNT100;
   1:  PR[GP1:91,1] = PR[GP1:90,1] + -22.134;
   1:  PR[GP1:91,2] = PR[GP1:90,2] + -40.812;
   1:L PR[91] 10mm/sec CNT100;
   1:  PR[GP1:91,1] = PR[GP1:90,1] + -10.660;
   1:  PR[GP1:91,2] = PR[GP1:90,2] + -42.071;
   1:L PR[91] 10mm/sec CNT100;
   1:  PR[GP1:91,1] = PR[GP1:90,1] + -7.295;
   1:  PR[GP1:91,2] = PR[GP1:90,2] + -41.507;
   1:L PR[91] 10mm/sec CNT100;
   1:  PR[GP1:91,1] = PR[GP1:90,1] + -0.262;
   1:  PR[GP1:91,2] = PR[GP1:90,2] + -39.995;
   1:L PR[91] 10mm/sec CNT100;
   1:  PR[GP1:91,1] = PR[GP1:90,1] + 6.333;
   1:  PR[GP1:91,2] = PR[GP1:90,2] + -41.594;
   1:  PR[GP1:91,3] = PR[GP1:90,3] + 95.465;
   1:L PR[91] 10mm/sec CNT100;
   1:  PR[GP1:91,1] = PR[GP1:90,1] + 9.943;
   1:  PR[GP1:91,2] = PR[GP1:90,2] + -42.200;
   1:L PR[91] 10mm/sec CNT100;
   1:  PR[GP1:91,1] = PR[GP1:90,1] + 21.206;
   1:  PR[GP1:91,2] = PR[GP1:90,2] + -40.963;
   1:L PR[91] 10mm/sec CNT100;
   1:  PR[GP1:91,1] = PR[GP1:90,1] + 24.415;
   1:  PR[GP1:91,2] = PR[GP1:90,2] + -40.363;
   1:L PR[91] 10mm/sec CNT100;
   1:  PR[GP1:91,1] = PR[GP1:90,1] + 35.034;
   1:  PR[GP1:91,2] = PR[GP1:90,2] + -35.516;
   1:L PR[91] 10mm/sec CNT100;
   1:  PR[GP1:91,1] = PR[GP1:90,1] + 37.281;
   1:  PR[GP1:91,2] = PR[GP1:90,2] + -34.124;
   1:L PR[91] 10mm/sec CNT100;
   1:  PR[GP1:91,1] = PR[GP1:90,1] + 46.016;
   1:  PR[GP1:91,2] = PR[GP1:90,2] + -26.005;
   1:L PR[91] 10mm/sec CNT100;
   1:  PR[GP1:91,1] = PR[GP1:90,1] + 47.011;
   1:  PR[GP1:91,2] = PR[GP1:90,2] + -24.806;
   1:L PR[91] 10mm/sec CNT100;
   1:  PR[GP1:91,1] = PR[GP1:90,1] + 52.813;
   1:  PR[GP1:91,2] = PR[GP1:90,2] + -14.130;
   1:L PR[91] 10mm/sec CNT100;
   1:  PR[GP1:91,1] = PR[GP1:90,1] + 53.331;
   1:  PR[GP1:91,2] = PR[GP1:90,2] + -12.958;
   1:L PR[91] 10mm/sec CNT100;
   1:  PR[GP1:91,1] = PR[GP1:90,1] + 55.352;
   1:  PR[GP1:91,2] = PR[GP1:90,2] + -0.929;
   1:L PR[91] 10mm/sec CNT100;
   1:  PR[GP1:91,1] = PR[GP1:90,1] + 55.356;
   1:  PR[GP1:91,2] = PR[GP1:90,2] + -0.634;
   1:L PR[91] 10mm/sec CNT100;
   1:  PR[GP1:91,1] = PR[GP1:90,1] + 55.482;
   1:  PR[GP1:91,2] = PR[GP1:90,2] + 0.271;
   1:L PR[91] 10mm/sec CNT100;
   1:  PR[GP1:91,1] = PR[GP1:90,1] + 53.499;
   1:  PR[GP1:91,2] = PR[GP1:90,2] + 12.255;
   1:L PR[91] 10mm/sec CNT100;
   1:  PR[GP1:91,1] = PR[GP1:90,1] + 53.319;
   1:  PR[GP1:91,2] = PR[GP1:90,2] + 13.548;
   1:L PR[91] 10mm/sec CNT100;
   1:  PR[GP1:91,1] = PR[GP1:90,1] + 52.805;
   1:  PR[GP1:91,2] = PR[GP1:90,2] + 14.712;
   1:L PR[91] 10mm/sec CNT100;
   1:  PR[GP1:91,1] = PR[GP1:90,1] + 46.979;
   1:  PR[GP1:91,2] = PR[GP1:90,2] + 25.405;
   1:L PR[91] 10mm/sec CNT100;
   1:  PR[GP1:91,1] = PR[GP1:90,1] + 45.983;
   1:  PR[GP1:91,2] = PR[GP1:90,2] + 26.604;
   1:L PR[91] 10mm/sec CNT100;
   1:  PR[GP1:91,1] = PR[GP1:90,1] + 37.219;
   1:  PR[GP1:91,2] = PR[GP1:90,2] + 34.723;
   1:L PR[91] 10mm/sec CNT100;
   1:  PR[GP1:91,1] = PR[GP1:90,1] + 34.969;
   1:  PR[GP1:91,2] = PR[GP1:90,2] + 36.117;
   1:L PR[91] 10mm/sec CNT100;
   1:  PR[GP1:91,1] = PR[GP1:90,1] + 24.322;
   1:  PR[GP1:91,2] = PR[GP1:90,2] + 40.947;
   1:L PR[91] 10mm/sec CNT100;
   1:  PR[GP1:91,1] = PR[GP1:90,1] + 21.108;
   1:  PR[GP1:91,2] = PR[GP1:90,2] + 41.547;
   1:L PR[91] 10mm/sec CNT100;
   1:  PR[GP1:91,1] = PR[GP1:90,1] + 9.829;
   1:  PR[GP1:91,2] = PR[GP1:90,2] + 42.752;
   1:L PR[91] 10mm/sec CNT100;
   1:  PR[GP1:91,1] = PR[GP1:90,1] + 4.751;
   1:  PR[GP1:91,2] = PR[GP1:90,2] + 41.859;
   1:L PR[91] 10mm/sec CNT100;
   1:  PR[GP1:91,1] = PR[GP1:90,1] + -0.260;
   1:  PR[GP1:91,2] = PR[GP1:90,2] + 40.766;
   1:L PR[91] 10mm/sec CNT100;
   1:  PR[GP1:91,1] = PR[GP1:90,1] + -5.273;
   1:  PR[GP1:91,2] = PR[GP1:90,2] + 41.859;
   1:L PR[91] 10mm/sec CNT100;
   1:  PR[GP1:91,1] = PR[GP1:90,1] + -10.356;
   1:  PR[GP1:91,2] = PR[GP1:90,2] + 42.752;
   1:L PR[91] 10mm/sec CNT100;
   1:  PR[GP1:91,1] = PR[GP1:90,1] + -21.635;
   1:  PR[GP1:91,2] = PR[GP1:90,2] + 41.548;
   1:L PR[91] 10mm/sec CNT100;
   1:  PR[GP1:91,1] = PR[GP1:90,1] + -24.848;
   1:  PR[GP1:91,2] = PR[GP1:90,2] + 40.947;
   1:L PR[91] 10mm/sec CNT100;
   1:  PR[GP1:91,1] = PR[GP1:90,1] + -35.495;
   1:  PR[GP1:91,2] = PR[GP1:90,2] + 36.114;
   1:L PR[91] 10mm/sec CNT100;
   1:  PR[GP1:91,1] = PR[GP1:90,1] + -37.745;
   1:  PR[GP1:91,2] = PR[GP1:90,2] + 34.721;
   1:L PR[91] 10mm/sec CNT100;
   1:  PR[GP1:91,1] = PR[GP1:90,1] + -46.509;
   1:  PR[GP1:91,2] = PR[GP1:90,2] + 26.611;
   1:L PR[91] 10mm/sec CNT100;
   1:  PR[GP1:91,1] = PR[GP1:90,1] + -47.505;
   1:  PR[GP1:91,2] = PR[GP1:90,2] + 25.412;
   1:L PR[91] 10mm/sec CNT100;
   1:  PR[GP1:91,1] = PR[GP1:90,1] + -53.331;
   1:  PR[GP1:91,2] = PR[GP1:90,2] + 14.700;
   1:L PR[91] 10mm/sec CNT100;
   1:  PR[GP1:91,1] = PR[GP1:90,1] + -53.849;
   1:  PR[GP1:91,2] = PR[GP1:90,2] + 13.527;
   1:L PR[91] 10mm/sec CNT100;
   1:  PR[GP1:91,1] = PR[GP1:90,1] + -55.879;
   1:  PR[GP1:91,2] = PR[GP1:90,2] + 1.487;
   1:L PR[91] 10mm/sec CNT100;
   1:  PR[GP1:91,1] = PR[GP1:90,1] + -55.882;
   1:  PR[GP1:91,2] = PR[GP1:90,2] + 1.192;
   1:L PR[91] 10mm/sec CNT100;
   1:  PR[GP1:91,1] = PR[GP1:90,1] + -56.008;
   1:  PR[GP1:91,2] = PR[GP1:90,2] + 0.287;
   1:L PR[91] 10mm/sec CNT100;
   1:  PR[GP1:91,1] = PR[GP1:90,1] + -54.034;
   1:  PR[GP1:91,2] = PR[GP1:90,2] + -11.660;
   1:L PR[91] 10mm/sec CNT100;
   1:  PR[GP1:91,1] = PR[GP1:90,1] + -53.854;
   1:  PR[GP1:91,2] = PR[GP1:90,2] + -12.953;
   1:L PR[91] 10mm/sec CNT100;
   1:  PR[GP1:91,1] = PR[GP1:90,1] + -53.340;
   1:  PR[GP1:91,2] = PR[GP1:90,2] + -14.117;
   1:L PR[91] 10mm/sec CNT100;
   1:  PR[GP1:91,1] = PR[GP1:90,1] + -47.537;
   1:  PR[GP1:91,2] = PR[GP1:90,2] + -24.813;
   1:L PR[91] 10mm/sec CNT100;
   1:  PR[GP1:91,1] = PR[GP1:90,1] + -46.542;
   1:  PR[GP1:91,2] = PR[GP1:90,2] + -26.012;
   1:L PR[91] 10mm/sec CNT100;
   1:  PR[GP1:91,1] = PR[GP1:90,1] + -37.807;
   1:  PR[GP1:91,2] = PR[GP1:90,2] + -34.122;
   1:L PR[91] 10mm/sec CNT100;
   1:  PR[GP1:91,1] = PR[GP1:90,1] + -35.561;
   1:  PR[GP1:91,2] = PR[GP1:90,2] + -35.513;
   1:L PR[91] 10mm/sec CNT100;
   1:  PR[GP1:91,1] = PR[GP1:90,1] + -24.942;
   1:  PR[GP1:91,2] = PR[GP1:90,2] + -40.364;
   1:L PR[91] 10mm/sec CNT100;
   1:  PR[GP1:91,1] = PR[GP1:90,1] + -21.734;
   1:  PR[GP1:91,2] = PR[GP1:90,2] + -40.964;
   1:L PR[91] 10mm/sec CNT100;
   1:  PR[GP1:91,1] = PR[GP1:90,1] + -10.471;
   1:  PR[GP1:91,2] = PR[GP1:90,2] + -42.200;
   1:L PR[91] 10mm/sec CNT100;
   1:  PR[GP1:91,1] = PR[GP1:90,1] + -6.857;
   1:  PR[GP1:91,2] = PR[GP1:90,2] + -41.594;
   1:L PR[91] 10mm/sec CNT100;
   1:  PR[GP1:91,1] = PR[GP1:90,1] + -0.262;
   1:  PR[GP1:91,2] = PR[GP1:90,2] + -40.176;
   1:L PR[91] 10mm/sec CNT100;
   1:  PR[GP1:91,1] = PR[GP1:90,1] + 5.895;
   1:  PR[GP1:91,2] = PR[GP1:90,2] + -41.681;
   1:  PR[GP1:91,3] = PR[GP1:90,3] + 96.075;
   1:L PR[91] 10mm/sec CNT100;
   1:  PR[GP1:91,1] = PR[GP1:90,1] + 9.754;
   1:  PR[GP1:91,2] = PR[GP1:90,2] + -42.329;
   1:L PR[91] 10mm/sec CNT100;
   1:  PR[GP1:91,1] = PR[GP1:90,1] + 20.806;
   1:  PR[GP1:91,2] = PR[GP1:90,2] + -41.115;
   1:L PR[91] 10mm/sec CNT100;
   1:  PR[GP1:91,1] = PR[GP1:90,1] + 24.289;
   1:  PR[GP1:91,2] = PR[GP1:90,2] + -40.463;
   1:L PR[91] 10mm/sec CNT100;
   1:  PR[GP1:91,1] = PR[GP1:90,1] + 34.709;
   1:  PR[GP1:91,2] = PR[GP1:90,2] + -35.707;
   1:L PR[91] 10mm/sec CNT100;
   1:  PR[GP1:91,1] = PR[GP1:90,1] + 37.203;
   1:  PR[GP1:91,2] = PR[GP1:90,2] + -34.163;
   1:L PR[91] 10mm/sec CNT100;
   1:  PR[GP1:91,1] = PR[GP1:90,1] + 45.774;
   1:  PR[GP1:91,2] = PR[GP1:90,2] + -26.195;
   1:L PR[91] 10mm/sec CNT100;
   1:  PR[GP1:91,1] = PR[GP1:90,1] + 46.913;
   1:  PR[GP1:91,2] = PR[GP1:90,2] + -24.822;
   1:L PR[91] 10mm/sec CNT100;
   1:  PR[GP1:91,1] = PR[GP1:90,1] + 52.607;
   1:  PR[GP1:91,2] = PR[GP1:90,2] + -14.346;
   1:L PR[91] 10mm/sec CNT100;
   1:  PR[GP1:91,1] = PR[GP1:90,1] + 53.218;
   1:  PR[GP1:91,2] = PR[GP1:90,2] + -12.963;
   1:L PR[91] 10mm/sec CNT100;
   1:  PR[GP1:91,1] = PR[GP1:90,1] + 55.202;
   1:  PR[GP1:91,2] = PR[GP1:90,2] + -1.160;
   1:L PR[91] 10mm/sec CNT100;
   1:  PR[GP1:91,1] = PR[GP1:90,1] + 55.205;
   1:  PR[GP1:91,2] = PR[GP1:90,2] + -0.870;
   1:L PR[91] 10mm/sec CNT100;
   1:  PR[GP1:91,1] = PR[GP1:90,1] + 55.364;
   1:  PR[GP1:91,2] = PR[GP1:90,2] + 0.271;
   1:L PR[91] 10mm/sec CNT100;
   1:  PR[GP1:91,1] = PR[GP1:90,1] + 53.418;
   1:  PR[GP1:91,2] = PR[GP1:90,2] + 12.031;
   1:L PR[91] 10mm/sec CNT100;
   1:  PR[GP1:91,1] = PR[GP1:90,1] + 53.206;
   1:  PR[GP1:91,2] = PR[GP1:90,2] + 13.553;
   1:L PR[91] 10mm/sec CNT100;
   1:  PR[GP1:91,1] = PR[GP1:90,1] + 52.599;
   1:  PR[GP1:91,2] = PR[GP1:90,2] + 14.928;
   1:L PR[91] 10mm/sec CNT100;
   1:  PR[GP1:91,1] = PR[GP1:90,1] + 46.882;
   1:  PR[GP1:91,2] = PR[GP1:90,2] + 25.420;
   1:L PR[91] 10mm/sec CNT100;
   1:  PR[GP1:91,1] = PR[GP1:90,1] + 45.742;
   1:  PR[GP1:91,2] = PR[GP1:90,2] + 26.794;
   1:L PR[91] 10mm/sec CNT100;
   1:  PR[GP1:91,1] = PR[GP1:90,1] + 37.142;
   1:  PR[GP1:91,2] = PR[GP1:90,2] + 34.761;
   1:L PR[91] 10mm/sec CNT100;
   1:  PR[GP1:91,1] = PR[GP1:90,1] + 34.645;
   1:  PR[GP1:91,2] = PR[GP1:90,2] + 36.307;
   1:L PR[91] 10mm/sec CNT100;
   1:  PR[GP1:91,1] = PR[GP1:90,1] + 24.198;
   1:  PR[GP1:91,2] = PR[GP1:90,2] + 41.047;
   1:L PR[91] 10mm/sec CNT100;
   1:  PR[GP1:91,1] = PR[GP1:90,1] + 20.709;
   1:  PR[GP1:91,2] = PR[GP1:90,2] + 41.699;
   1:L PR[91] 10mm/sec CNT100;
   1:  PR[GP1:91,1] = PR[GP1:90,1] + 9.642;
   1:  PR[GP1:91,2] = PR[GP1:90,2] + 42.881;
   1:L PR[91] 10mm/sec CNT100;
   1:  PR[GP1:91,1] = PR[GP1:90,1] + 4.218;
   1:  PR[GP1:91,2] = PR[GP1:90,2] + 41.926;
   1:L PR[91] 10mm/sec CNT100;
   1:  PR[GP1:91,1] = PR[GP1:90,1] + -0.260;
   1:  PR[GP1:91,2] = PR[GP1:90,2] + 40.950;
   1:L PR[91] 10mm/sec CNT100;
   1:  PR[GP1:91,1] = PR[GP1:90,1] + -4.739;
   1:  PR[GP1:91,2] = PR[GP1:90,2] + 41.926;
   1:L PR[91] 10mm/sec CNT100;
   1:  PR[GP1:91,1] = PR[GP1:90,1] + -10.169;
   1:  PR[GP1:91,2] = PR[GP1:90,2] + 42.880;
   1:L PR[91] 10mm/sec CNT100;
   1:  PR[GP1:91,1] = PR[GP1:90,1] + -21.237;
   1:  PR[GP1:91,2] = PR[GP1:90,2] + 41.700;
   1:L PR[91] 10mm/sec CNT100;
   1:  PR[GP1:91,1] = PR[GP1:90,1] + -24.724;
   1:  PR[GP1:91,2] = PR[GP1:90,2] + 41.047;
   1:L PR[91] 10mm/sec CNT100;
   1:  PR[GP1:91,1] = PR[GP1:90,1] + -35.171;
   1:  PR[GP1:91,2] = PR[GP1:90,2] + 36.305;
   1:L PR[91] 10mm/sec CNT100;
   1:  PR[GP1:91,1] = PR[GP1:90,1] + -37.668;
   1:  PR[GP1:91,2] = PR[GP1:90,2] + 34.759;
   1:L PR[91] 10mm/sec CNT100;
   1:  PR[GP1:91,1] = PR[GP1:90,1] + -46.268;
   1:  PR[GP1:91,2] = PR[GP1:90,2] + 26.801;
   1:L PR[91] 10mm/sec CNT100;
   1:  PR[GP1:91,1] = PR[GP1:90,1] + -47.408;
   1:  PR[GP1:91,2] = PR[GP1:90,2] + 25.428;
   1:L PR[91] 10mm/sec CNT100;
   1:  PR[GP1:91,1] = PR[GP1:90,1] + -53.125;
   1:  PR[GP1:91,2] = PR[GP1:90,2] + 14.916;
   1:L PR[91] 10mm/sec CNT100;
   1:  PR[GP1:91,1] = PR[GP1:90,1] + -53.736;
   1:  PR[GP1:91,2] = PR[GP1:90,2] + 13.532;
   1:L PR[91] 10mm/sec CNT100;
   1:  PR[GP1:91,1] = PR[GP1:90,1] + -55.728;
   1:  PR[GP1:91,2] = PR[GP1:90,2] + 1.718;
   1:L PR[91] 10mm/sec CNT100;
   1:  PR[GP1:91,1] = PR[GP1:90,1] + -55.731;
   1:  PR[GP1:91,2] = PR[GP1:90,2] + 1.428;
   1:L PR[91] 10mm/sec CNT100;
   1:  PR[GP1:91,1] = PR[GP1:90,1] + -55.890;
   1:  PR[GP1:91,2] = PR[GP1:90,2] + 0.287;
   1:L PR[91] 10mm/sec CNT100;
   1:  PR[GP1:91,1] = PR[GP1:90,1] + -53.953;
   1:  PR[GP1:91,2] = PR[GP1:90,2] + -11.437;
   1:L PR[91] 10mm/sec CNT100;
   1:  PR[GP1:91,1] = PR[GP1:90,1] + -53.741;
   1:  PR[GP1:91,2] = PR[GP1:90,2] + -12.958;
   1:L PR[91] 10mm/sec CNT100;
   1:  PR[GP1:91,1] = PR[GP1:90,1] + -53.133;
   1:  PR[GP1:91,2] = PR[GP1:90,2] + -14.334;
   1:L PR[91] 10mm/sec CNT100;
   1:  PR[GP1:91,1] = PR[GP1:90,1] + -47.439;
   1:  PR[GP1:91,2] = PR[GP1:90,2] + -24.829;
   1:L PR[91] 10mm/sec CNT100;
   1:  PR[GP1:91,1] = PR[GP1:90,1] + -46.300;
   1:  PR[GP1:91,2] = PR[GP1:90,2] + -26.202;
   1:L PR[91] 10mm/sec CNT100;
   1:  PR[GP1:91,1] = PR[GP1:90,1] + -37.729;
   1:  PR[GP1:91,2] = PR[GP1:90,2] + -34.160;
   1:L PR[91] 10mm/sec CNT100;
   1:  PR[GP1:91,1] = PR[GP1:90,1] + -35.236;
   1:  PR[GP1:91,2] = PR[GP1:90,2] + -35.704;
   1:L PR[91] 10mm/sec CNT100;
   1:  PR[GP1:91,1] = PR[GP1:90,1] + -24.816;
   1:  PR[GP1:91,2] = PR[GP1:90,2] + -40.464;
   1:L PR[91] 10mm/sec CNT100;
   1:  PR[GP1:91,1] = PR[GP1:90,1] + -21.334;
   1:  PR[GP1:91,2] = PR[GP1:90,2] + -41.116;
   1:L PR[91] 10mm/sec CNT100;
   1:  PR[GP1:91,1] = PR[GP1:90,1] + -10.282;
   1:  PR[GP1:91,2] = PR[GP1:90,2] + -42.328;
   1:L PR[91] 10mm/sec CNT100;
   1:  PR[GP1:91,1] = PR[GP1:90,1] + -6.419;
   1:  PR[GP1:91,2] = PR[GP1:90,2] + -41.681;
   1:L PR[91] 10mm/sec CNT100;
   1:  PR[GP1:91,1] = PR[GP1:90,1] + -0.262;
   1:  PR[GP1:91,2] = PR[GP1:90,2] + -40.357;
   1:L PR[91] 10mm/sec CNT100;
   1:  PR[GP1:91,1] = PR[GP1:90,1] + 5.457;
   1:  PR[GP1:91,2] = PR[GP1:90,2] + -41.768;
   1:  PR[GP1:91,3] = PR[GP1:90,3] + 96.685;
   1:L PR[91] 10mm/sec CNT100;
   1:  PR[GP1:91,1] = PR[GP1:90,1] + 9.564;
   1:  PR[GP1:91,2] = PR[GP1:90,2] + -42.457;
   1:L PR[91] 10mm/sec CNT100;
   1:  PR[GP1:91,1] = PR[GP1:90,1] + 20.405;
   1:  PR[GP1:91,2] = PR[GP1:90,2] + -41.266;
   1:L PR[91] 10mm/sec CNT100;
   1:  PR[GP1:91,1] = PR[GP1:90,1] + 24.163;
   1:  PR[GP1:91,2] = PR[GP1:90,2] + -40.564;
   1:L PR[91] 10mm/sec CNT100;
   1:  PR[GP1:91,1] = PR[GP1:90,1] + 34.383;
   1:  PR[GP1:91,2] = PR[GP1:90,2] + -35.898;
   1:L PR[91] 10mm/sec CNT100;
   1:  PR[GP1:91,1] = PR[GP1:90,1] + 37.124;
   1:  PR[GP1:91,2] = PR[GP1:90,2] + -34.201;
   1:L PR[91] 10mm/sec CNT100;
   1:  PR[GP1:91,1] = PR[GP1:90,1] + 45.532;
   1:  PR[GP1:91,2] = PR[GP1:90,2] + -26.385;
   1:L PR[91] 10mm/sec CNT100;
   1:  PR[GP1:91,1] = PR[GP1:90,1] + 46.816;
   1:  PR[GP1:91,2] = PR[GP1:90,2] + -24.839;
   1:L PR[91] 10mm/sec CNT100;
   1:  PR[GP1:91,1] = PR[GP1:90,1] + 52.401;
   1:  PR[GP1:91,2] = PR[GP1:90,2] + -14.562;
   1:L PR[91] 10mm/sec CNT100;
   1:  PR[GP1:91,1] = PR[GP1:90,1] + 53.105;
   1:  PR[GP1:91,2] = PR[GP1:90,2] + -12.968;
   1:L PR[91] 10mm/sec CNT100;
   1:  PR[GP1:91,1] = PR[GP1:90,1] + 55.051;
   1:  PR[GP1:91,2] = PR[GP1:90,2] + -1.391;
   1:L PR[91] 10mm/sec CNT100;
   1:  PR[GP1:91,1] = PR[GP1:90,1] + 55.054;
   1:  PR[GP1:91,2] = PR[GP1:90,2] + -1.106;
   1:L PR[91] 10mm/sec CNT100;
   1:  PR[GP1:91,1] = PR[GP1:90,1] + 55.246;
   1:  PR[GP1:91,2] = PR[GP1:90,2] + 0.271;
   1:L PR[91] 10mm/sec CNT100;
   1:  PR[GP1:91,1] = PR[GP1:90,1] + 53.337;
   1:  PR[GP1:91,2] = PR[GP1:90,2] + 11.807;
   1:L PR[91] 10mm/sec CNT100;
   1:  PR[GP1:91,1] = PR[GP1:90,1] + 53.093;
   1:  PR[GP1:91,2] = PR[GP1:90,2] + 13.557;
   1:L PR[91] 10mm/sec CNT100;
   1:  PR[GP1:91,1] = PR[GP1:90,1] + 52.393;
   1:  PR[GP1:91,2] = PR[GP1:90,2] + 15.144;
   1:L PR[91] 10mm/sec CNT100;
   1:  PR[GP1:91,1] = PR[GP1:90,1] + 46.785;
   1:  PR[GP1:91,2] = PR[GP1:90,2] + 25.436;
   1:L PR[91] 10mm/sec CNT100;
   1:  PR[GP1:91,1] = PR[GP1:90,1] + 45.501;
   1:  PR[GP1:91,2] = PR[GP1:90,2] + 26.984;
   1:L PR[91] 10mm/sec CNT100;
   1:  PR[GP1:91,1] = PR[GP1:90,1] + 37.064;
   1:  PR[GP1:91,2] = PR[GP1:90,2] + 34.798;
   1:L PR[91] 10mm/sec CNT100;
   1:  PR[GP1:91,1] = PR[GP1:90,1] + 34.321;
   1:  PR[GP1:91,2] = PR[GP1:90,2] + 36.498;
   1:L PR[91] 10mm/sec CNT100;
   1:  PR[GP1:91,1] = PR[GP1:90,1] + 24.073;
   1:  PR[GP1:91,2] = PR[GP1:90,2] + 41.146;
   1:L PR[91] 10mm/sec CNT100;
   1:  PR[GP1:91,1] = PR[GP1:90,1] + 20.310;
   1:  PR[GP1:91,2] = PR[GP1:90,2] + 41.850;
   1:L PR[91] 10mm/sec CNT100;
   1:  PR[GP1:91,1] = PR[GP1:90,1] + 9.454;
   1:  PR[GP1:91,2] = PR[GP1:90,2] + 43.009;
   1:L PR[91] 10mm/sec CNT100;
   1:  PR[GP1:91,1] = PR[GP1:90,1] + 3.684;
   1:  PR[GP1:91,2] = PR[GP1:90,2] + 41.994;
   1:L PR[91] 10mm/sec CNT100;
   1:  PR[GP1:91,1] = PR[GP1:90,1] + -0.260;
   1:  PR[GP1:91,2] = PR[GP1:90,2] + 41.134;
   1:L PR[91] 10mm/sec CNT100;
   1:  PR[GP1:91,1] = PR[GP1:90,1] + -4.205;
   1:  PR[GP1:91,2] = PR[GP1:90,2] + 41.994;
   1:L PR[91] 10mm/sec CNT100;
   1:  PR[GP1:91,1] = PR[GP1:90,1] + -9.982;
   1:  PR[GP1:91,2] = PR[GP1:90,2] + 43.009;
   1:L PR[91] 10mm/sec CNT100;
   1:  PR[GP1:91,1] = PR[GP1:90,1] + -20.838;
   1:  PR[GP1:91,2] = PR[GP1:90,2] + 41.851;
   1:L PR[91] 10mm/sec CNT100;
   1:  PR[GP1:91,1] = PR[GP1:90,1] + -24.600;
   1:  PR[GP1:91,2] = PR[GP1:90,2] + 41.147;
   1:L PR[91] 10mm/sec CNT100;
   1:  PR[GP1:91,1] = PR[GP1:90,1] + -34.847;
   1:  PR[GP1:91,2] = PR[GP1:90,2] + 36.495;
   1:L PR[91] 10mm/sec CNT100;
   1:  PR[GP1:91,1] = PR[GP1:90,1] + -37.590;
   1:  PR[GP1:91,2] = PR[GP1:90,2] + 34.796;
   1:L PR[91] 10mm/sec CNT100;
   1:  PR[GP1:91,1] = PR[GP1:90,1] + -46.027;
   1:  PR[GP1:91,2] = PR[GP1:90,2] + 26.990;
   1:L PR[91] 10mm/sec CNT100;
   1:  PR[GP1:91,1] = PR[GP1:90,1] + -47.311;
   1:  PR[GP1:91,2] = PR[GP1:90,2] + 25.443;
   1:L PR[91] 10mm/sec CNT100;
   1:  PR[GP1:91,1] = PR[GP1:90,1] + -52.919;
   1:  PR[GP1:91,2] = PR[GP1:90,2] + 15.132;
   1:L PR[91] 10mm/sec CNT100;
   1:  PR[GP1:91,1] = PR[GP1:90,1] + -53.623;
   1:  PR[GP1:91,2] = PR[GP1:90,2] + 13.537;
   1:L PR[91] 10mm/sec CNT100;
   1:  PR[GP1:91,1] = PR[GP1:90,1] + -55.577;
   1:  PR[GP1:91,2] = PR[GP1:90,2] + 1.949;
   1:L PR[91] 10mm/sec CNT100;
   1:  PR[GP1:91,1] = PR[GP1:90,1] + -55.580;
   1:  PR[GP1:91,2] = PR[GP1:90,2] + 1.665;
   1:L PR[91] 10mm/sec CNT100;
   1:  PR[GP1:91,1] = PR[GP1:90,1] + -55.772;
   1:  PR[GP1:91,2] = PR[GP1:90,2] + 0.287;
   1:L PR[91] 10mm/sec CNT100;
   1:  PR[GP1:91,1] = PR[GP1:90,1] + -53.872;
   1:  PR[GP1:91,2] = PR[GP1:90,2] + -11.213;
   1:L PR[91] 10mm/sec CNT100;
   1:  PR[GP1:91,1] = PR[GP1:90,1] + -53.628;
   1:  PR[GP1:91,2] = PR[GP1:90,2] + -12.963;
   1:L PR[91] 10mm/sec CNT100;
   1:  PR[GP1:91,1] = PR[GP1:90,1] + -52.927;
   1:  PR[GP1:91,2] = PR[GP1:90,2] + -14.550;
   1:L PR[91] 10mm/sec CNT100;
   1:  PR[GP1:91,1] = PR[GP1:90,1] + -47.342;
   1:  PR[GP1:91,2] = PR[GP1:90,2] + -24.846;
   1:L PR[91] 10mm/sec CNT100;
   1:  PR[GP1:91,1] = PR[GP1:90,1] + -46.058;
   1:  PR[GP1:91,2] = PR[GP1:90,2] + -26.392;
   1:L PR[91] 10mm/sec CNT100;
   1:  PR[GP1:91,1] = PR[GP1:90,1] + -37.651;
   1:  PR[GP1:91,2] = PR[GP1:90,2] + -34.198;
   1:L PR[91] 10mm/sec CNT100;
   1:  PR[GP1:91,1] = PR[GP1:90,1] + -34.910;
   1:  PR[GP1:91,2] = PR[GP1:90,2] + -35.896;
   1:L PR[91] 10mm/sec CNT100;
   1:  PR[GP1:91,1] = PR[GP1:90,1] + -24.690;
   1:  PR[GP1:91,2] = PR[GP1:90,2] + -40.565;
   1:L PR[91] 10mm/sec CNT100;
   1:  PR[GP1:91,1] = PR[GP1:90,1] + -20.933;
   1:  PR[GP1:91,2] = PR[GP1:90,2] + -41.267;
   1:L PR[91] 10mm/sec CNT100;
   1:  PR[GP1:91,1] = PR[GP1:90,1] + -10.093;
   1:  PR[GP1:91,2] = PR[GP1:90,2] + -42.457;
   1:L PR[91] 10mm/sec CNT100;
   1:  PR[GP1:91,1] = PR[GP1:90,1] + -5.981;
   1:  PR[GP1:91,2] = PR[GP1:90,2] + -41.767;
   1:L PR[91] 10mm/sec CNT100;
   1:  PR[GP1:91,1] = PR[GP1:90,1] + -0.262;
   1:  PR[GP1:91,2] = PR[GP1:90,2] + -40.538;
   1:L PR[91] 10mm/sec CNT100;
   1:  PR[GP1:91,1] = PR[GP1:90,1] + 5.020;
   1:  PR[GP1:91,2] = PR[GP1:90,2] + -41.854;
   1:  PR[GP1:91,3] = PR[GP1:90,3] + 97.295;
   1:L PR[91] 10mm/sec CNT100;
   1:  PR[GP1:91,1] = PR[GP1:90,1] + 9.375;
   1:  PR[GP1:91,2] = PR[GP1:90,2] + -42.586;
   1:L PR[91] 10mm/sec CNT100;
   1:  PR[GP1:91,1] = PR[GP1:90,1] + 20.005;
   1:  PR[GP1:91,2] = PR[GP1:90,2] + -41.418;
   1:L PR[91] 10mm/sec CNT100;
   1:  PR[GP1:91,1] = PR[GP1:90,1] + 24.037;
   1:  PR[GP1:91,2] = PR[GP1:90,2] + -40.664;
   1:L PR[91] 10mm/sec CNT100;
   1:  PR[GP1:91,1] = PR[GP1:90,1] + 34.058;
   1:  PR[GP1:91,2] = PR[GP1:90,2] + -36.090;
   1:L PR[91] 10mm/sec CNT100;
   1:  PR[GP1:91,1] = PR[GP1:90,1] + 37.046;
   1:  PR[GP1:91,2] = PR[GP1:90,2] + -34.239;
   1:L PR[91] 10mm/sec CNT100;
   1:  PR[GP1:91,1] = PR[GP1:90,1] + 45.290;
   1:  PR[GP1:91,2] = PR[GP1:90,2] + -26.576;
   1:L PR[91] 10mm/sec CNT100;
   1:  PR[GP1:91,1] = PR[GP1:90,1] + 46.718;
   1:  PR[GP1:91,2] = PR[GP1:90,2] + -24.856;
   1:L PR[91] 10mm/sec CNT100;
   1:  PR[GP1:91,1] = PR[GP1:90,1] + 52.195;
   1:  PR[GP1:91,2] = PR[GP1:90,2] + -14.778;
   1:L PR[91] 10mm/sec CNT100;
   1:  PR[GP1:91,1] = PR[GP1:90,1] + 52.992;
   1:  PR[GP1:91,2] = PR[GP1:90,2] + -12.973;
   1:L PR[91] 10mm/sec CNT100;
   1:  PR[GP1:91,1] = PR[GP1:90,1] + 54.900;
   1:  PR[GP1:91,2] = PR[GP1:90,2] + -1.621;
   1:L PR[91] 10mm/sec CNT100;
   1:  PR[GP1:91,1] = PR[GP1:90,1] + 54.903;
   1:  PR[GP1:91,2] = PR[GP1:90,2] + -1.343;
   1:L PR[91] 10mm/sec CNT100;
   1:  PR[GP1:91,1] = PR[GP1:90,1] + 55.128;
   1:  PR[GP1:91,2] = PR[GP1:90,2] + 0.271;
   1:L PR[91] 10mm/sec CNT100;
   1:  PR[GP1:91,1] = PR[GP1:90,1] + 53.256;
   1:  PR[GP1:91,2] = PR[GP1:90,2] + 11.583;
   1:L PR[91] 10mm/sec CNT100;
   1:  PR[GP1:91,1] = PR[GP1:90,1] + 52.980;
   1:  PR[GP1:91,2] = PR[GP1:90,2] + 13.562;
   1:L PR[91] 10mm/sec CNT100;
   1:  PR[GP1:91,1] = PR[GP1:90,1] + 52.187;
   1:  PR[GP1:91,2] = PR[GP1:90,2] + 15.360;
   1:L PR[91] 10mm/sec CNT100;
   1:  PR[GP1:91,1] = PR[GP1:90,1] + 46.688;
   1:  PR[GP1:91,2] = PR[GP1:90,2] + 25.452;
   1:L PR[91] 10mm/sec CNT100;
   1:  PR[GP1:91,1] = PR[GP1:90,1] + 45.259;
   1:  PR[GP1:91,2] = PR[GP1:90,2] + 27.173;
   1:L PR[91] 10mm/sec CNT100;
   1:  PR[GP1:91,1] = PR[GP1:90,1] + 36.987;
   1:  PR[GP1:91,2] = PR[GP1:90,2] + 34.836;
   1:L PR[91] 10mm/sec CNT100;
   1:  PR[GP1:91,1] = PR[GP1:90,1] + 33.996;
   1:  PR[GP1:91,2] = PR[GP1:90,2] + 36.688;
   1:L PR[91] 10mm/sec CNT100;
   1:  PR[GP1:91,1] = PR[GP1:90,1] + 23.949;
   1:  PR[GP1:91,2] = PR[GP1:90,2] + 41.246;
   1:L PR[91] 10mm/sec CNT100;
   1:  PR[GP1:91,1] = PR[GP1:90,1] + 19.912;
   1:  PR[GP1:91,2] = PR[GP1:90,2] + 42.001;
   1:L PR[91] 10mm/sec CNT100;
   1:  PR[GP1:91,1] = PR[GP1:90,1] + 9.267;
   1:  PR[GP1:91,2] = PR[GP1:90,2] + 43.138;
   1:L PR[91] 10mm/sec CNT100;
   1:  PR[GP1:91,1] = PR[GP1:90,1] + 3.151;
   1:  PR[GP1:91,2] = PR[GP1:90,2] + 42.062;
   1:L PR[91] 10mm/sec CNT100;
   1:  PR[GP1:91,1] = PR[GP1:90,1] + -0.260;
   1:  PR[GP1:91,2] = PR[GP1:90,2] + 41.318;
   1:L PR[91] 10mm/sec CNT100;
   1:  PR[GP1:91,1] = PR[GP1:90,1] + -3.671;
   1:  PR[GP1:91,2] = PR[GP1:90,2] + 42.062;
   1:L PR[91] 10mm/sec CNT100;
   1:  PR[GP1:91,1] = PR[GP1:90,1] + -9.795;
   1:  PR[GP1:91,2] = PR[GP1:90,2] + 43.137;
   1:L PR[91] 10mm/sec CNT100;
   1:  PR[GP1:91,1] = PR[GP1:90,1] + -20.440;
   1:  PR[GP1:91,2] = PR[GP1:90,2] + 42.002;
   1:L PR[91] 10mm/sec CNT100;
   1:  PR[GP1:91,1] = PR[GP1:90,1] + -24.475;
   1:  PR[GP1:91,2] = PR[GP1:90,2] + 41.247;
   1:L PR[91] 10mm/sec CNT100;
   1:  PR[GP1:91,1] = PR[GP1:90,1] + -34.523;
   1:  PR[GP1:91,2] = PR[GP1:90,2] + 36.686;
   1:L PR[91] 10mm/sec CNT100;
   1:  PR[GP1:91,1] = PR[GP1:90,1] + -37.513;
   1:  PR[GP1:91,2] = PR[GP1:90,2] + 34.834;
   1:L PR[91] 10mm/sec CNT100;
   1:  PR[GP1:91,1] = PR[GP1:90,1] + -45.785;
   1:  PR[GP1:91,2] = PR[GP1:90,2] + 27.180;
   1:L PR[91] 10mm/sec CNT100;
   1:  PR[GP1:91,1] = PR[GP1:90,1] + -47.214;
   1:  PR[GP1:91,2] = PR[GP1:90,2] + 25.459;
   1:L PR[91] 10mm/sec CNT100;
   1:  PR[GP1:91,1] = PR[GP1:90,1] + -52.713;
   1:  PR[GP1:91,2] = PR[GP1:90,2] + 15.348;
   1:L PR[91] 10mm/sec CNT100;
   1:  PR[GP1:91,1] = PR[GP1:90,1] + -53.510;
   1:  PR[GP1:91,2] = PR[GP1:90,2] + 13.542;
   1:L PR[91] 10mm/sec CNT100;
   1:  PR[GP1:91,1] = PR[GP1:90,1] + -55.426;
   1:  PR[GP1:91,2] = PR[GP1:90,2] + 2.179;
   1:L PR[91] 10mm/sec CNT100;
   1:  PR[GP1:91,1] = PR[GP1:90,1] + -55.429;
   1:  PR[GP1:91,2] = PR[GP1:90,2] + 1.901;
   1:L PR[91] 10mm/sec CNT100;
   1:  PR[GP1:91,1] = PR[GP1:90,1] + -55.654;
   1:  PR[GP1:91,2] = PR[GP1:90,2] + 0.287;
   1:L PR[91] 10mm/sec CNT100;
   1:  PR[GP1:91,1] = PR[GP1:90,1] + -53.791;
   1:  PR[GP1:91,2] = PR[GP1:90,2] + -10.990;
   1:L PR[91] 10mm/sec CNT100;
   1:  PR[GP1:91,1] = PR[GP1:90,1] + -53.515;
   1:  PR[GP1:91,2] = PR[GP1:90,2] + -12.968;
   1:L PR[91] 10mm/sec CNT100;
   1:  PR[GP1:91,1] = PR[GP1:90,1] + -52.721;
   1:  PR[GP1:91,2] = PR[GP1:90,2] + -14.767;
   1:L PR[91] 10mm/sec CNT100;
   1:  PR[GP1:91,1] = PR[GP1:90,1] + -47.244;
   1:  PR[GP1:91,2] = PR[GP1:90,2] + -24.862;
   1:L PR[91] 10mm/sec CNT100;
   1:  PR[GP1:91,1] = PR[GP1:90,1] + -45.816;
   1:  PR[GP1:91,2] = PR[GP1:90,2] + -26.582;
   1:L PR[91] 10mm/sec CNT100;
   1:  PR[GP1:91,1] = PR[GP1:90,1] + -37.572;
   1:  PR[GP1:91,2] = PR[GP1:90,2] + -34.237;
   1:L PR[91] 10mm/sec CNT100;
   1:  PR[GP1:91,1] = PR[GP1:90,1] + -34.585;
   1:  PR[GP1:91,2] = PR[GP1:90,2] + -36.087;
   1:L PR[91] 10mm/sec CNT100;
   1:  PR[GP1:91,1] = PR[GP1:90,1] + -24.564;
   1:  PR[GP1:91,2] = PR[GP1:90,2] + -40.665;
   1:L PR[91] 10mm/sec CNT100;
   1:  PR[GP1:91,1] = PR[GP1:90,1] + -20.533;
   1:  PR[GP1:91,2] = PR[GP1:90,2] + -41.419;
   1:L PR[91] 10mm/sec CNT100;
   1:  PR[GP1:91,1] = PR[GP1:90,1] + -9.903;
   1:  PR[GP1:91,2] = PR[GP1:90,2] + -42.585;
   1:L PR[91] 10mm/sec CNT100;
   1:  PR[GP1:91,1] = PR[GP1:90,1] + -5.543;
   1:  PR[GP1:91,2] = PR[GP1:90,2] + -41.854;
   1:L PR[91] 10mm/sec CNT100;
   1:  PR[GP1:91,1] = PR[GP1:90,1] + -0.262;
   1:  PR[GP1:91,2] = PR[GP1:90,2] + -40.719;
   1:L PR[91] 10mm/sec CNT100;
   1:  PR[GP1:91,1] = PR[GP1:90,1] + 4.582;
   1:  PR[GP1:91,2] = PR[GP1:90,2] + -41.941;
   1:  PR[GP1:91,3] = PR[GP1:90,3] + 97.905;
   1:L PR[91] 10mm/sec CNT100;
   1:  PR[GP1:91,1] = PR[GP1:90,1] + 9.186;
   1:  PR[GP1:91,2] = PR[GP1:90,2] + -42.714;
   1:L PR[91] 10mm/sec CNT100;
   1:  PR[GP1:91,1] = PR[GP1:90,1] + 19.604;
   1:  PR[GP1:91,2] = PR[GP1:90,2] + -41.570;
   1:L PR[91] 10mm/sec CNT100;
   1:  PR[GP1:91,1] = PR[GP1:90,1] + 23.910;
   1:  PR[GP1:91,2] = PR[GP1:90,2] + -40.765;
   1:L PR[91] 10mm/sec CNT100;
   1:  PR[GP1:91,1] = PR[GP1:90,1] + 33.733;
   1:  PR[GP1:91,2] = PR[GP1:90,2] + -36.281;
   1:L PR[91] 10mm/sec CNT100;
   1:  PR[GP1:91,1] = PR[GP1:90,1] + 36.968;
   1:  PR[GP1:91,2] = PR[GP1:90,2] + -34.277;
   1:L PR[91] 10mm/sec CNT100;
   1:  PR[GP1:91,1] = PR[GP1:90,1] + 45.048;
   1:  PR[GP1:91,2] = PR[GP1:90,2] + -26.766;
   1:L PR[91] 10mm/sec CNT100;
   1:  PR[GP1:91,1] = PR[GP1:90,1] + 46.620;
   1:  PR[GP1:91,2] = PR[GP1:90,2] + -24.872;
   1:L PR[91] 10mm/sec CNT100;
   1:  PR[GP1:91,1] = PR[GP1:90,1] + 51.989;
   1:  PR[GP1:91,2] = PR[GP1:90,2] + -14.995;
   1:L PR[91] 10mm/sec CNT100;
   1:  PR[GP1:91,1] = PR[GP1:90,1] + 52.879;
   1:  PR[GP1:91,2] = PR[GP1:90,2] + -12.978;
   1:L PR[91] 10mm/sec CNT100;
   1:  PR[GP1:91,1] = PR[GP1:90,1] + 54.749;
   1:  PR[GP1:91,2] = PR[GP1:90,2] + -1.852;
   1:L PR[91] 10mm/sec CNT100;
   1:  PR[GP1:91,1] = PR[GP1:90,1] + 54.752;
   1:  PR[GP1:91,2] = PR[GP1:90,2] + -1.579;
   1:L PR[91] 10mm/sec CNT100;
   1:  PR[GP1:91,1] = PR[GP1:90,1] + 55.010;
   1:  PR[GP1:91,2] = PR[GP1:90,2] + 0.271;
   1:L PR[91] 10mm/sec CNT100;
   1:  PR[GP1:91,1] = PR[GP1:90,1] + 53.175;
   1:  PR[GP1:91,2] = PR[GP1:90,2] + 11.359;
   1:L PR[91] 10mm/sec CNT100;
   1:  PR[GP1:91,1] = PR[GP1:90,1] + 52.868;
   1:  PR[GP1:91,2] = PR[GP1:90,2] + 13.566;
   1:L PR[91] 10mm/sec CNT100;
   1:  PR[GP1:91,1] = PR[GP1:90,1] + 51.981;
   1:  PR[GP1:91,2] = PR[GP1:90,2] + 15.576;
   1:L PR[91] 10mm/sec CNT100;
   1:  PR[GP1:91,1] = PR[GP1:90,1] + 46.591;
   1:  PR[GP1:91,2] = PR[GP1:90,2] + 25.468;
   1:L PR[91] 10mm/sec CNT100;
   1:  PR[GP1:91,1] = PR[GP1:90,1] + 45.018;
   1:  PR[GP1:91,2] = PR[GP1:90,2] + 27.363;
   1:L PR[91] 10mm/sec CNT100;
   1:  PR[GP1:91,1] = PR[GP1:90,1] + 36.910;
   1:  PR[GP1:91,2] = PR[GP1:90,2] + 34.873;
   1:L PR[91] 10mm/sec CNT100;
   1:  PR[GP1:91,1] = PR[GP1:90,1] + 33.672;
   1:  PR[GP1:91,2] = PR[GP1:90,2] + 36.879;
   1:L PR[91] 10mm/sec CNT100;
   1:  PR[GP1:91,1] = PR[GP1:90,1] + 23.824;
   1:  PR[GP1:91,2] = PR[GP1:90,2] + 41.346;
   1:L PR[91] 10mm/sec CNT100;
   1:  PR[GP1:91,1] = PR[GP1:90,1] + 19.513;
   1:  PR[GP1:91,2] = PR[GP1:90,2] + 42.152;
   1:L PR[91] 10mm/sec CNT100;
   1:  PR[GP1:91,1] = PR[GP1:90,1] + 9.080;
   1:  PR[GP1:91,2] = PR[GP1:90,2] + 43.266;
   1:L PR[91] 10mm/sec CNT100;
   1:  PR[GP1:91,1] = PR[GP1:90,1] + 2.617;
   1:  PR[GP1:91,2] = PR[GP1:90,2] + 42.129;
   1:L PR[91] 10mm/sec CNT100;
   1:  PR[GP1:91,1] = PR[GP1:90,1] + -0.260;
   1:  PR[GP1:91,2] = PR[GP1:90,2] + 41.502;
   1:L PR[91] 10mm/sec CNT100;
   1:  PR[GP1:91,1] = PR[GP1:90,1] + -3.138;
   1:  PR[GP1:91,2] = PR[GP1:90,2] + 42.129;
   1:L PR[91] 10mm/sec CNT100;
   1:  PR[GP1:91,1] = PR[GP1:90,1] + -9.608;
   1:  PR[GP1:91,2] = PR[GP1:90,2] + 43.266;
   1:L PR[91] 10mm/sec CNT100;
   1:  PR[GP1:91,1] = PR[GP1:90,1] + -20.041;
   1:  PR[GP1:91,2] = PR[GP1:90,2] + 42.153;
   1:L PR[91] 10mm/sec CNT100;
   1:  PR[GP1:91,1] = PR[GP1:90,1] + -24.351;
   1:  PR[GP1:91,2] = PR[GP1:90,2] + 41.347;
   1:L PR[91] 10mm/sec CNT100;
   1:  PR[GP1:91,1] = PR[GP1:90,1] + -34.199;
   1:  PR[GP1:91,2] = PR[GP1:90,2] + 36.876;
   1:L PR[91] 10mm/sec CNT100;
   1:  PR[GP1:91,1] = PR[GP1:90,1] + -37.436;
   1:  PR[GP1:91,2] = PR[GP1:90,2] + 34.871;
   1:L PR[91] 10mm/sec CNT100;
   1:  PR[GP1:91,1] = PR[GP1:90,1] + -45.544;
   1:  PR[GP1:91,2] = PR[GP1:90,2] + 27.369;
   1:L PR[91] 10mm/sec CNT100;
   1:  PR[GP1:91,1] = PR[GP1:90,1] + -47.117;
   1:  PR[GP1:91,2] = PR[GP1:90,2] + 25.475;
   1:L PR[91] 10mm/sec CNT100;
   1:  PR[GP1:91,1] = PR[GP1:90,1] + -52.507;
   1:  PR[GP1:91,2] = PR[GP1:90,2] + 15.564;
   1:L PR[91] 10mm/sec CNT100;
   1:  PR[GP1:91,1] = PR[GP1:90,1] + -53.397;
   1:  PR[GP1:91,2] = PR[GP1:90,2] + 13.547;
   1:L PR[91] 10mm/sec CNT100;
   1:  PR[GP1:91,1] = PR[GP1:90,1] + -55.275;
   1:  PR[GP1:91,2] = PR[GP1:90,2] + 2.410;
   1:L PR[91] 10mm/sec CNT100;
   1:  PR[GP1:91,1] = PR[GP1:90,1] + -55.278;
   1:  PR[GP1:91,2] = PR[GP1:90,2] + 2.137;
   1:L PR[91] 10mm/sec CNT100;
   1:  PR[GP1:91,1] = PR[GP1:90,1] + -55.536;
   1:  PR[GP1:91,2] = PR[GP1:90,2] + 0.287;
   1:L PR[91] 10mm/sec CNT100;
   1:  PR[GP1:91,1] = PR[GP1:90,1] + -53.710;
   1:  PR[GP1:91,2] = PR[GP1:90,2] + -10.766;
   1:L PR[91] 10mm/sec CNT100;
   1:  PR[GP1:91,1] = PR[GP1:90,1] + -53.402;
   1:  PR[GP1:91,2] = PR[GP1:90,2] + -12.974;
   1:L PR[91] 10mm/sec CNT100;
   1:  PR[GP1:91,1] = PR[GP1:90,1] + -52.515;
   1:  PR[GP1:91,2] = PR[GP1:90,2] + -14.983;
   1:L PR[91] 10mm/sec CNT100;
   1:  PR[GP1:91,1] = PR[GP1:90,1] + -47.146;
   1:  PR[GP1:91,2] = PR[GP1:90,2] + -24.879;
   1:L PR[91] 10mm/sec CNT100;
   1:  PR[GP1:91,1] = PR[GP1:90,1] + -45.574;
   1:  PR[GP1:91,2] = PR[GP1:90,2] + -26.773;
   1:L PR[91] 10mm/sec CNT100;
   1:  PR[GP1:91,1] = PR[GP1:90,1] + -37.494;
   1:  PR[GP1:91,2] = PR[GP1:90,2] + -34.275;
   1:L PR[91] 10mm/sec CNT100;
   1:  PR[GP1:91,1] = PR[GP1:90,1] + -34.260;
   1:  PR[GP1:91,2] = PR[GP1:90,2] + -36.278;
   1:L PR[91] 10mm/sec CNT100;
   1:  PR[GP1:91,1] = PR[GP1:90,1] + -24.438;
   1:  PR[GP1:91,2] = PR[GP1:90,2] + -40.765;
   1:L PR[91] 10mm/sec CNT100;
   1:  PR[GP1:91,1] = PR[GP1:90,1] + -20.133;
   1:  PR[GP1:91,2] = PR[GP1:90,2] + -41.570;
   1:L PR[91] 10mm/sec CNT100;
   1:  PR[GP1:91,1] = PR[GP1:90,1] + -9.714;
   1:  PR[GP1:91,2] = PR[GP1:90,2] + -42.714;
   1:L PR[91] 10mm/sec CNT100;
   1:  PR[GP1:91,1] = PR[GP1:90,1] + -5.105;
   1:  PR[GP1:91,2] = PR[GP1:90,2] + -41.941;
   1:L PR[91] 10mm/sec CNT100;
   1:  PR[GP1:91,1] = PR[GP1:90,1] + -0.261;
   1:  PR[GP1:91,2] = PR[GP1:90,2] + -40.899;
   1:L PR[91] 10mm/sec CNT100;
   1:  PR[GP1:91,1] = PR[GP1:90,1] + 4.144;
   1:  PR[GP1:91,2] = PR[GP1:90,2] + -42.028;
   1:  PR[GP1:91,3] = PR[GP1:90,3] + 98.515;
   1:L PR[91] 10mm/sec CNT100;
   1:  PR[GP1:91,1] = PR[GP1:90,1] + 8.996;
   1:  PR[GP1:91,2] = PR[GP1:90,2] + -42.843;
   1:L PR[91] 10mm/sec CNT100;
   1:  PR[GP1:91,1] = PR[GP1:90,1] + 19.204;
   1:  PR[GP1:91,2] = PR[GP1:90,2] + -41.721;
   1:L PR[91] 10mm/sec CNT100;
   1:  PR[GP1:91,1] = PR[GP1:90,1] + 23.784;
   1:  PR[GP1:91,2] = PR[GP1:90,2] + -40.865;
   1:L PR[91] 10mm/sec CNT100;
   1:  PR[GP1:91,1] = PR[GP1:90,1] + 33.407;
   1:  PR[GP1:91,2] = PR[GP1:90,2] + -36.472;
   1:L PR[91] 10mm/sec CNT100;
   1:  PR[GP1:91,1] = PR[GP1:90,1] + 36.889;
   1:  PR[GP1:91,2] = PR[GP1:90,2] + -34.316;
   1:L PR[91] 10mm/sec CNT100;
   1:  PR[GP1:91,1] = PR[GP1:90,1] + 44.806;
   1:  PR[GP1:91,2] = PR[GP1:90,2] + -26.956;
   1:L PR[91] 10mm/sec CNT100;
   1:  PR[GP1:91,1] = PR[GP1:90,1] + 46.522;
   1:  PR[GP1:91,2] = PR[GP1:90,2] + -24.889;
   1:L PR[91] 10mm/sec CNT100;
   1:  PR[GP1:91,1] = PR[GP1:90,1] + 51.782;
   1:  PR[GP1:91,2] = PR[GP1:90,2] + -15.211;
   1:L PR[91] 10mm/sec CNT100;
   1:  PR[GP1:91,1] = PR[GP1:90,1] + 52.766;
   1:  PR[GP1:91,2] = PR[GP1:90,2] + -12.983;
   1:L PR[91] 10mm/sec CNT100;
   1:  PR[GP1:91,1] = PR[GP1:90,1] + 54.598;
   1:  PR[GP1:91,2] = PR[GP1:90,2] + -2.083;
   1:L PR[91] 10mm/sec CNT100;
   1:  PR[GP1:91,1] = PR[GP1:90,1] + 54.601;
   1:  PR[GP1:91,2] = PR[GP1:90,2] + -1.815;
   1:L PR[91] 10mm/sec CNT100;
   1:  PR[GP1:91,1] = PR[GP1:90,1] + 54.892;
   1:  PR[GP1:91,2] = PR[GP1:90,2] + 0.271;
   1:L PR[91] 10mm/sec CNT100;
   1:  PR[GP1:91,1] = PR[GP1:90,1] + 53.095;
   1:  PR[GP1:91,2] = PR[GP1:90,2] + 11.134;
   1:L PR[91] 10mm/sec CNT100;
   1:  PR[GP1:91,1] = PR[GP1:90,1] + 52.755;
   1:  PR[GP1:91,2] = PR[GP1:90,2] + 13.571;
   1:L PR[91] 10mm/sec CNT100;
   1:  PR[GP1:91,1] = PR[GP1:90,1] + 51.775;
   1:  PR[GP1:91,2] = PR[GP1:90,2] + 15.791;
   1:L PR[91] 10mm/sec CNT100;
   1:  PR[GP1:91,1] = PR[GP1:90,1] + 46.494;
   1:  PR[GP1:91,2] = PR[GP1:90,2] + 25.484;
   1:L PR[91] 10mm/sec CNT100;
   1:  PR[GP1:91,1] = PR[GP1:90,1] + 44.777;
   1:  PR[GP1:91,2] = PR[GP1:90,2] + 27.552;
   1:L PR[91] 10mm/sec CNT100;
   1:  PR[GP1:91,1] = PR[GP1:90,1] + 36.833;
   1:  PR[GP1:91,2] = PR[GP1:90,2] + 34.911;
   1:L PR[91] 10mm/sec CNT100;
   1:  PR[GP1:91,1] = PR[GP1:90,1] + 33.348;
   1:  PR[GP1:91,2] = PR[GP1:90,2] + 37.069;
   1:L PR[91] 10mm/sec CNT100;
   1:  PR[GP1:91,1] = PR[GP1:90,1] + 23.700;
   1:  PR[GP1:91,2] = PR[GP1:90,2] + 41.446;
   1:L PR[91] 10mm/sec CNT100;
   1:  PR[GP1:91,1] = PR[GP1:90,1] + 19.114;
   1:  PR[GP1:91,2] = PR[GP1:90,2] + 42.303;
   1:L PR[91] 10mm/sec CNT100;
   1:  PR[GP1:91,1] = PR[GP1:90,1] + 8.893;
   1:  PR[GP1:91,2] = PR[GP1:90,2] + 43.395;
   1:L PR[91] 10mm/sec CNT100;
   1:  PR[GP1:91,1] = PR[GP1:90,1] + 2.084;
   1:  PR[GP1:91,2] = PR[GP1:90,2] + 42.197;
   1:L PR[91] 10mm/sec CNT100;
   1:  PR[GP1:91,1] = PR[GP1:90,1] + -0.260;
   1:  PR[GP1:91,2] = PR[GP1:90,2] + 41.686;
   1:L PR[91] 10mm/sec CNT100;
   1:  PR[GP1:91,1] = PR[GP1:90,1] + -2.604;
   1:  PR[GP1:91,2] = PR[GP1:90,2] + 42.197;
   1:L PR[91] 10mm/sec CNT100;
   1:  PR[GP1:91,1] = PR[GP1:90,1] + -9.421;
   1:  PR[GP1:91,2] = PR[GP1:90,2] + 43.394;
   1:L PR[91] 10mm/sec CNT100;
   1:  PR[GP1:91,1] = PR[GP1:90,1] + -19.642;
   1:  PR[GP1:91,2] = PR[GP1:90,2] + 42.304;
   1:L PR[91] 10mm/sec CNT100;
   1:  PR[GP1:91,1] = PR[GP1:90,1] + -24.226;
   1:  PR[GP1:91,2] = PR[GP1:90,2] + 41.447;
   1:L PR[91] 10mm/sec CNT100;
   1:  PR[GP1:91,1] = PR[GP1:90,1] + -33.875;
   1:  PR[GP1:91,2] = PR[GP1:90,2] + 37.067;
   1:L PR[91] 10mm/sec CNT100;
   1:  PR[GP1:91,1] = PR[GP1:90,1] + -37.359;
   1:  PR[GP1:91,2] = PR[GP1:90,2] + 34.909;
   1:L PR[91] 10mm/sec CNT100;
   1:  PR[GP1:91,1] = PR[GP1:90,1] + -45.303;
   1:  PR[GP1:91,2] = PR[GP1:90,2] + 27.559;
   1:L PR[91] 10mm/sec CNT100;
   1:  PR[GP1:91,1] = PR[GP1:90,1] + -47.020;
   1:  PR[GP1:91,2] = PR[GP1:90,2] + 25.490;
   1:L PR[91] 10mm/sec CNT100;
   1:  PR[GP1:91,1] = PR[GP1:90,1] + -52.301;
   1:  PR[GP1:91,2] = PR[GP1:90,2] + 15.780;
   1:L PR[91] 10mm/sec CNT100;
   1:  PR[GP1:91,1] = PR[GP1:90,1] + -53.285;
   1:  PR[GP1:91,2] = PR[GP1:90,2] + 13.552;
   1:L PR[91] 10mm/sec CNT100;
   1:  PR[GP1:91,1] = PR[GP1:90,1] + -55.124;
   1:  PR[GP1:91,2] = PR[GP1:90,2] + 2.641;
   1:L PR[91] 10mm/sec CNT100;
   1:  PR[GP1:91,1] = PR[GP1:90,1] + -55.127;
   1:  PR[GP1:91,2] = PR[GP1:90,2] + 2.374;
   1:L PR[91] 10mm/sec CNT100;
   1:  PR[GP1:91,1] = PR[GP1:90,1] + -55.418;
   1:  PR[GP1:91,2] = PR[GP1:90,2] + 0.287;
   1:L PR[91] 10mm/sec CNT100;
   1:  PR[GP1:91,1] = PR[GP1:90,1] + -53.629;
   1:  PR[GP1:91,2] = PR[GP1:90,2] + -10.543;
   1:L PR[91] 10mm/sec CNT100;
   1:  PR[GP1:91,1] = PR[GP1:90,1] + -53.289;
   1:  PR[GP1:91,2] = PR[GP1:90,2] + -12.979;
   1:L PR[91] 10mm/sec CNT100;
   1:  PR[GP1:91,1] = PR[GP1:90,1] + -52.309;
   1:  PR[GP1:91,2] = PR[GP1:90,2] + -15.200;
   1:L PR[91] 10mm/sec CNT100;
   1:  PR[GP1:91,1] = PR[GP1:90,1] + -47.049;
   1:  PR[GP1:91,2] = PR[GP1:90,2] + -24.895;
   1:L PR[91] 10mm/sec CNT100;
   1:  PR[GP1:91,1] = PR[GP1:90,1] + -45.332;
   1:  PR[GP1:91,2] = PR[GP1:90,2] + -26.963;
   1:L PR[91] 10mm/sec CNT100;
   1:  PR[GP1:91,1] = PR[GP1:90,1] + -37.416;
   1:  PR[GP1:91,2] = PR[GP1:90,2] + -34.313;
   1:L PR[91] 10mm/sec CNT100;
   1:  PR[GP1:91,1] = PR[GP1:90,1] + -33.934;
   1:  PR[GP1:91,2] = PR[GP1:90,2] + -36.470;
   1:L PR[91] 10mm/sec CNT100;
   1:  PR[GP1:91,1] = PR[GP1:90,1] + -24.311;
   1:  PR[GP1:91,2] = PR[GP1:90,2] + -40.866;
   1:L PR[91] 10mm/sec CNT100;
   1:  PR[GP1:91,1] = PR[GP1:90,1] + -19.732;
   1:  PR[GP1:91,2] = PR[GP1:90,2] + -41.722;
   1:L PR[91] 10mm/sec CNT100;
   1:  PR[GP1:91,1] = PR[GP1:90,1] + -9.525;
   1:  PR[GP1:91,2] = PR[GP1:90,2] + -42.842;
   1:L PR[91] 10mm/sec CNT100;
   1:  PR[GP1:91,1] = PR[GP1:90,1] + -4.667;
   1:  PR[GP1:91,2] = PR[GP1:90,2] + -42.028;
   1:L PR[91] 10mm/sec CNT100;
   1:  PR[GP1:91,1] = PR[GP1:90,1] + -0.261;
   1:  PR[GP1:91,2] = PR[GP1:90,2] + -41.080;
   1:L PR[91] 10mm/sec CNT100;
   1:  PR[GP1:91,1] = PR[GP1:90,1] + 3.706;
   1:  PR[GP1:91,2] = PR[GP1:90,2] + -42.115;
   1:  PR[GP1:91,3] = PR[GP1:90,3] + 99.125;
   1:L PR[91] 10mm/sec CNT100;
   1:  PR[GP1:91,1] = PR[GP1:90,1] + 8.807;
   1:  PR[GP1:91,2] = PR[GP1:90,2] + -42.971;
   1:L PR[91] 10mm/sec CNT100;
   1:  PR[GP1:91,1] = PR[GP1:90,1] + 18.803;
   1:  PR[GP1:91,2] = PR[GP1:90,2] + -41.873;
   1:L PR[91] 10mm/sec CNT100;
   1:  PR[GP1:91,1] = PR[GP1:90,1] + 23.658;
   1:  PR[GP1:91,2] = PR[GP1:90,2] + -40.965;
   1:L PR[91] 10mm/sec CNT100;
   1:  PR[GP1:91,1] = PR[GP1:90,1] + 33.082;
   1:  PR[GP1:91,2] = PR[GP1:90,2] + -36.663;
   1:L PR[91] 10mm/sec CNT100;
   1:  PR[GP1:91,1] = PR[GP1:90,1] + 36.811;
   1:  PR[GP1:91,2] = PR[GP1:90,2] + -34.354;
   1:L PR[91] 10mm/sec CNT100;
   1:  PR[GP1:91,1] = PR[GP1:90,1] + 44.564;
   1:  PR[GP1:91,2] = PR[GP1:90,2] + -27.147;
   1:L PR[91] 10mm/sec CNT100;
   1:  PR[GP1:91,1] = PR[GP1:90,1] + 46.425;
   1:  PR[GP1:91,2] = PR[GP1:90,2] + -24.905;
   1:L PR[91] 10mm/sec CNT100;
   1:  PR[GP1:91,1] = PR[GP1:90,1] + 51.576;
   1:  PR[GP1:91,2] = PR[GP1:90,2] + -15.427;
   1:L PR[91] 10mm/sec CNT100;
   1:  PR[GP1:91,1] = PR[GP1:90,1] + 52.653;
   1:  PR[GP1:91,2] = PR[GP1:90,2] + -12.988;
   1:L PR[91] 10mm/sec CNT100;
   1:  PR[GP1:91,1] = PR[GP1:90,1] + 54.447;
   1:  PR[GP1:91,2] = PR[GP1:90,2] + -2.313;
   1:L PR[91] 10mm/sec CNT100;
   1:  PR[GP1:91,1] = PR[GP1:90,1] + 54.450;
   1:  PR[GP1:91,2] = PR[GP1:90,2] + -2.052;
   1:L PR[91] 10mm/sec CNT100;
   1:  PR[GP1:91,1] = PR[GP1:90,1] + 54.774;
   1:  PR[GP1:91,2] = PR[GP1:90,2] + 0.271;
   1:L PR[91] 10mm/sec CNT100;
   1:  PR[GP1:91,1] = PR[GP1:90,1] + 53.014;
   1:  PR[GP1:91,2] = PR[GP1:90,2] + 10.910;
   1:L PR[91] 10mm/sec CNT100;
   1:  PR[GP1:91,1] = PR[GP1:90,1] + 52.642;
   1:  PR[GP1:91,2] = PR[GP1:90,2] + 13.575;
   1:L PR[91] 10mm/sec CNT100;
   1:  PR[GP1:91,1] = PR[GP1:90,1] + 51.568;
   1:  PR[GP1:91,2] = PR[GP1:90,2] + 16.007;
   1:L PR[91] 10mm/sec CNT100;
   1:  PR[GP1:91,1] = PR[GP1:90,1] + 46.397;
   1:  PR[GP1:91,2] = PR[GP1:90,2] + 25.500;
   1:L PR[91] 10mm/sec CNT100;
   1:  PR[GP1:91,1] = PR[GP1:90,1] + 44.535;
   1:  PR[GP1:91,2] = PR[GP1:90,2] + 27.742;
   1:L PR[91] 10mm/sec CNT100;
   1:  PR[GP1:91,1] = PR[GP1:90,1] + 36.756;
   1:  PR[GP1:91,2] = PR[GP1:90,2] + 34.949;
   1:L PR[91] 10mm/sec CNT100;
   1:  PR[GP1:91,1] = PR[GP1:90,1] + 33.024;
   1:  PR[GP1:91,2] = PR[GP1:90,2] + 37.260;
   1:L PR[91] 10mm/sec CNT100;
   1:  PR[GP1:91,1] = PR[GP1:90,1] + 23.575;
   1:  PR[GP1:91,2] = PR[GP1:90,2] + 41.546;
   1:L PR[91] 10mm/sec CNT100;
   1:  PR[GP1:91,1] = PR[GP1:90,1] + 18.716;
   1:  PR[GP1:91,2] = PR[GP1:90,2] + 42.454;
   1:L PR[91] 10mm/sec CNT100;
   1:  PR[GP1:91,1] = PR[GP1:90,1] + 8.706;
   1:  PR[GP1:91,2] = PR[GP1:90,2] + 43.523;
   1:L PR[91] 10mm/sec CNT100;
   1:  PR[GP1:91,1] = PR[GP1:90,1] + 1.550;
   1:  PR[GP1:91,2] = PR[GP1:90,2] + 42.265;
   1:L PR[91] 10mm/sec CNT100;
   1:  PR[GP1:91,1] = PR[GP1:90,1] + -0.260;
   1:  PR[GP1:91,2] = PR[GP1:90,2] + 41.870;
   1:L PR[91] 10mm/sec CNT100;
   1:  PR[GP1:91,1] = PR[GP1:90,1] + -2.070;
   1:  PR[GP1:91,2] = PR[GP1:90,2] + 42.265;
   1:L PR[91] 10mm/sec CNT100;
   1:  PR[GP1:91,1] = PR[GP1:90,1] + -9.234;
   1:  PR[GP1:91,2] = PR[GP1:90,2] + 43.523;
   1:L PR[91] 10mm/sec CNT100;
   1:  PR[GP1:91,1] = PR[GP1:90,1] + -19.244;
   1:  PR[GP1:91,2] = PR[GP1:90,2] + 42.455;
   1:L PR[91] 10mm/sec CNT100;
   1:  PR[GP1:91,1] = PR[GP1:90,1] + -24.102;
   1:  PR[GP1:91,2] = PR[GP1:90,2] + 41.547;
   1:L PR[91] 10mm/sec CNT100;
   1:  PR[GP1:91,1] = PR[GP1:90,1] + -33.551;
   1:  PR[GP1:91,2] = PR[GP1:90,2] + 37.257;
   1:L PR[91] 10mm/sec CNT100;
   1:  PR[GP1:91,1] = PR[GP1:90,1] + -37.282;
   1:  PR[GP1:91,2] = PR[GP1:90,2] + 34.947;
   1:L PR[91] 10mm/sec CNT100;
   1:  PR[GP1:91,1] = PR[GP1:90,1] + -45.061;
   1:  PR[GP1:91,2] = PR[GP1:90,2] + 27.748;
   1:L PR[91] 10mm/sec CNT100;
   1:  PR[GP1:91,1] = PR[GP1:90,1] + -46.923;
   1:  PR[GP1:91,2] = PR[GP1:90,2] + 25.506;
   1:L PR[91] 10mm/sec CNT100;
   1:  PR[GP1:91,1] = PR[GP1:90,1] + -52.095;
   1:  PR[GP1:91,2] = PR[GP1:90,2] + 15.996;
   1:L PR[91] 10mm/sec CNT100;
   1:  PR[GP1:91,1] = PR[GP1:90,1] + -53.172;
   1:  PR[GP1:91,2] = PR[GP1:90,2] + 13.556;
   1:L PR[91] 10mm/sec CNT100;
   1:  PR[GP1:91,1] = PR[GP1:90,1] + -54.973;
   1:  PR[GP1:91,2] = PR[GP1:90,2] + 2.871;
   1:L PR[91] 10mm/sec CNT100;
   1:  PR[GP1:91,1] = PR[GP1:90,1] + -54.976;
   1:  PR[GP1:91,2] = PR[GP1:90,2] + 2.610;
   1:L PR[91] 10mm/sec CNT100;
   1:  PR[GP1:91,1] = PR[GP1:90,1] + -55.300;
   1:  PR[GP1:91,2] = PR[GP1:90,2] + 0.287;
   1:L PR[91] 10mm/sec CNT100;
   1:  PR[GP1:91,1] = PR[GP1:90,1] + -53.548;
   1:  PR[GP1:91,2] = PR[GP1:90,2] + -10.319;
   1:L PR[91] 10mm/sec CNT100;
   1:  PR[GP1:91,1] = PR[GP1:90,1] + -53.176;
   1:  PR[GP1:91,2] = PR[GP1:90,2] + -12.984;
   1:L PR[91] 10mm/sec CNT100;
   1:  PR[GP1:91,1] = PR[GP1:90,1] + -52.102;
   1:  PR[GP1:91,2] = PR[GP1:90,2] + -15.416;
   1:L PR[91] 10mm/sec CNT100;
   1:  PR[GP1:91,1] = PR[GP1:90,1] + -46.951;
   1:  PR[GP1:91,2] = PR[GP1:90,2] + -24.912;
   1:L PR[91] 10mm/sec CNT100;
   1:  PR[GP1:91,1] = PR[GP1:90,1] + -45.090;
   1:  PR[GP1:91,2] = PR[GP1:90,2] + -27.153;
   1:L PR[91] 10mm/sec CNT100;
   1:  PR[GP1:91,1] = PR[GP1:90,1] + -37.337;
   1:  PR[GP1:91,2] = PR[GP1:90,2] + -34.352;
   1:L PR[91] 10mm/sec CNT100;
   1:  PR[GP1:91,1] = PR[GP1:90,1] + -33.609;
   1:  PR[GP1:91,2] = PR[GP1:90,2] + -36.661;
   1:L PR[91] 10mm/sec CNT100;
   1:  PR[GP1:91,1] = PR[GP1:90,1] + -24.185;
   1:  PR[GP1:91,2] = PR[GP1:90,2] + -40.966;
   1:L PR[91] 10mm/sec CNT100;
   1:  PR[GP1:91,1] = PR[GP1:90,1] + -19.332;
   1:  PR[GP1:91,2] = PR[GP1:90,2] + -41.874;
   1:L PR[91] 10mm/sec CNT100;
   1:  PR[GP1:91,1] = PR[GP1:90,1] + -9.336;
   1:  PR[GP1:91,2] = PR[GP1:90,2] + -42.971;
   1:L PR[91] 10mm/sec CNT100;
   1:  PR[GP1:91,1] = PR[GP1:90,1] + -4.229;
   1:  PR[GP1:91,2] = PR[GP1:90,2] + -42.114;
   1:L PR[91] 10mm/sec CNT100;
   1:  PR[GP1:91,1] = PR[GP1:90,1] + -0.261;
   1:  PR[GP1:91,2] = PR[GP1:90,2] + -41.261;
   1:L PR[91] 10mm/sec CNT100;
   1:  PR[GP1:91,1] = PR[GP1:90,1] + 3.268;
   1:  PR[GP1:91,2] = PR[GP1:90,2] + -42.201;
   1:  PR[GP1:91,3] = PR[GP1:90,3] + 99.735;
   1:L PR[91] 10mm/sec CNT100;
   1:  PR[GP1:91,1] = PR[GP1:90,1] + 8.618;
   1:  PR[GP1:91,2] = PR[GP1:90,2] + -43.099;
   1:L PR[91] 10mm/sec CNT100;
   1:  PR[GP1:91,1] = PR[GP1:90,1] + 18.403;
   1:  PR[GP1:91,2] = PR[GP1:90,2] + -42.024;
   1:L PR[91] 10mm/sec CNT100;
   1:  PR[GP1:91,1] = PR[GP1:90,1] + 23.532;
   1:  PR[GP1:91,2] = PR[GP1:90,2] + -41.066;
   1:L PR[91] 10mm/sec CNT100;
   1:  PR[GP1:91,1] = PR[GP1:90,1] + 32.757;
   1:  PR[GP1:91,2] = PR[GP1:90,2] + -36.855;
   1:L PR[91] 10mm/sec CNT100;
   1:  PR[GP1:91,1] = PR[GP1:90,1] + 36.733;
   1:  PR[GP1:91,2] = PR[GP1:90,2] + -34.392;
   1:L PR[91] 10mm/sec CNT100;
   1:  PR[GP1:91,1] = PR[GP1:90,1] + 44.322;
   1:  PR[GP1:91,2] = PR[GP1:90,2] + -27.337;
   1:L PR[91] 10mm/sec CNT100;
   1:  PR[GP1:91,1] = PR[GP1:90,1] + 46.327;
   1:  PR[GP1:91,2] = PR[GP1:90,2] + -24.922;
   1:L PR[91] 10mm/sec CNT100;
   1:  PR[GP1:91,1] = PR[GP1:90,1] + 51.370;
   1:  PR[GP1:91,2] = PR[GP1:90,2] + -15.644;
   1:L PR[91] 10mm/sec CNT100;
   1:  PR[GP1:91,1] = PR[GP1:90,1] + 52.540;
   1:  PR[GP1:91,2] = PR[GP1:90,2] + -12.993;
   1:L PR[91] 10mm/sec CNT100;
   1:  PR[GP1:91,1] = PR[GP1:90,1] + 54.296;
   1:  PR[GP1:91,2] = PR[GP1:90,2] + -2.544;
   1:L PR[91] 10mm/sec CNT100;
   1:  PR[GP1:91,1] = PR[GP1:90,1] + 54.299;
   1:  PR[GP1:91,2] = PR[GP1:90,2] + -2.288;
   1:L PR[91] 10mm/sec CNT100;
   1:  PR[GP1:91,1] = PR[GP1:90,1] + 54.656;
   1:  PR[GP1:91,2] = PR[GP1:90,2] + 0.271;
   1:L PR[91] 10mm/sec CNT100;
   1:  PR[GP1:91,1] = PR[GP1:90,1] + 52.933;
   1:  PR[GP1:91,2] = PR[GP1:90,2] + 10.686;
   1:L PR[91] 10mm/sec CNT100;
   1:  PR[GP1:91,1] = PR[GP1:90,1] + 52.529;
   1:  PR[GP1:91,2] = PR[GP1:90,2] + 13.580;
   1:L PR[91] 10mm/sec CNT100;
   1:  PR[GP1:91,1] = PR[GP1:90,1] + 51.362;
   1:  PR[GP1:91,2] = PR[GP1:90,2] + 16.223;
   1:L PR[91] 10mm/sec CNT100;
   1:  PR[GP1:91,1] = PR[GP1:90,1] + 46.300;
   1:  PR[GP1:91,2] = PR[GP1:90,2] + 25.515;
   1:L PR[91] 10mm/sec CNT100;
   1:  PR[GP1:91,1] = PR[GP1:90,1] + 44.294;
   1:  PR[GP1:91,2] = PR[GP1:90,2] + 27.931;
   1:L PR[91] 10mm/sec CNT100;
   1:  PR[GP1:91,1] = PR[GP1:90,1] + 36.678;
   1:  PR[GP1:91,2] = PR[GP1:90,2] + 34.986;
   1:L PR[91] 10mm/sec CNT100;
   1:  PR[GP1:91,1] = PR[GP1:90,1] + 32.700;
   1:  PR[GP1:91,2] = PR[GP1:90,2] + 37.450;
   1:L PR[91] 10mm/sec CNT100;
   1:  PR[GP1:91,1] = PR[GP1:90,1] + 23.451;
   1:  PR[GP1:91,2] = PR[GP1:90,2] + 41.646;
   1:L PR[91] 10mm/sec CNT100;
   1:  PR[GP1:91,1] = PR[GP1:90,1] + 18.317;
   1:  PR[GP1:91,2] = PR[GP1:90,2] + 42.605;
   1:L PR[91] 10mm/sec CNT100;
   1:  PR[GP1:91,1] = PR[GP1:90,1] + 8.519;
   1:  PR[GP1:91,2] = PR[GP1:90,2] + 43.652;
   1:L PR[91] 10mm/sec CNT100;
   1:  PR[GP1:91,1] = PR[GP1:90,1] + 1.017;
   1:  PR[GP1:91,2] = PR[GP1:90,2] + 42.332;
   1:L PR[91] 10mm/sec CNT100;
   1:  PR[GP1:91,1] = PR[GP1:90,1] + -0.260;
   1:  PR[GP1:91,2] = PR[GP1:90,2] + 42.054;
   1:L PR[91] 10mm/sec CNT100;
   1:  PR[GP1:91,1] = PR[GP1:90,1] + -1.537;
   1:  PR[GP1:91,2] = PR[GP1:90,2] + 42.332;
   1:L PR[91] 10mm/sec CNT100;
   1:  PR[GP1:91,1] = PR[GP1:90,1] + -9.047;
   1:  PR[GP1:91,2] = PR[GP1:90,2] + 43.652;
   1:L PR[91] 10mm/sec CNT100;
   1:  PR[GP1:91,1] = PR[GP1:90,1] + -18.845;
   1:  PR[GP1:91,2] = PR[GP1:90,2] + 42.606;
   1:L PR[91] 10mm/sec CNT100;
   1:  PR[GP1:91,1] = PR[GP1:90,1] + -23.977;
   1:  PR[GP1:91,2] = PR[GP1:90,2] + 41.647;
   1:L PR[91] 10mm/sec CNT100;
   1:  PR[GP1:91,1] = PR[GP1:90,1] + -33.227;
   1:  PR[GP1:91,2] = PR[GP1:90,2] + 37.448;
   1:L PR[91] 10mm/sec CNT100;
   1:  PR[GP1:91,1] = PR[GP1:90,1] + -37.204;
   1:  PR[GP1:91,2] = PR[GP1:90,2] + 34.984;
   1:L PR[91] 10mm/sec CNT100;
   1:  PR[GP1:91,1] = PR[GP1:90,1] + -44.820;
   1:  PR[GP1:91,2] = PR[GP1:90,2] + 27.938;
   1:L PR[91] 10mm/sec CNT100;
   1:  PR[GP1:91,1] = PR[GP1:90,1] + -46.826;
   1:  PR[GP1:91,2] = PR[GP1:90,2] + 25.522;
   1:L PR[91] 10mm/sec CNT100;
   1:  PR[GP1:91,1] = PR[GP1:90,1] + -51.889;
   1:  PR[GP1:91,2] = PR[GP1:90,2] + 16.212;
   1:L PR[91] 10mm/sec CNT100;
   1:  PR[GP1:91,1] = PR[GP1:90,1] + -53.059;
   1:  PR[GP1:91,2] = PR[GP1:90,2] + 13.561;
   1:L PR[91] 10mm/sec CNT100;
   1:  PR[GP1:91,1] = PR[GP1:90,1] + -54.823;
   1:  PR[GP1:91,2] = PR[GP1:90,2] + 3.102;
   1:L PR[91] 10mm/sec CNT100;
   1:  PR[GP1:91,1] = PR[GP1:90,1] + -54.825;
   1:  PR[GP1:91,2] = PR[GP1:90,2] + 2.846;
   1:L PR[91] 10mm/sec CNT100;
   1:  PR[GP1:91,1] = PR[GP1:90,1] + -55.182;
   1:  PR[GP1:91,2] = PR[GP1:90,2] + 0.287;
   1:L PR[91] 10mm/sec CNT100;
   1:  PR[GP1:91,1] = PR[GP1:90,1] + -53.467;
   1:  PR[GP1:91,2] = PR[GP1:90,2] + -10.096;
   1:L PR[91] 10mm/sec CNT100;
   1:  PR[GP1:91,1] = PR[GP1:90,1] + -53.063;
   1:  PR[GP1:91,2] = PR[GP1:90,2] + -12.990;
   1:L PR[91] 10mm/sec CNT100;
   1:  PR[GP1:91,1] = PR[GP1:90,1] + -51.896;
   1:  PR[GP1:91,2] = PR[GP1:90,2] + -15.633;
   1:L PR[91] 10mm/sec CNT100;
   1:  PR[GP1:91,1] = PR[GP1:90,1] + -46.853;
   1:  PR[GP1:91,2] = PR[GP1:90,2] + -24.928;
   1:L PR[91] 10mm/sec CNT100;
   1:  PR[GP1:91,1] = PR[GP1:90,1] + -44.848;
   1:  PR[GP1:91,2] = PR[GP1:90,2] + -27.343;
   1:L PR[91] 10mm/sec CNT100;
   1:  PR[GP1:91,1] = PR[GP1:90,1] + -37.259;
   1:  PR[GP1:91,2] = PR[GP1:90,2] + -34.390;
   1:L PR[91] 10mm/sec CNT100;
   1:  PR[GP1:91,1] = PR[GP1:90,1] + -33.284;
   1:  PR[GP1:91,2] = PR[GP1:90,2] + -36.852;
   1:L PR[91] 10mm/sec CNT100;
   1:  PR[GP1:91,1] = PR[GP1:90,1] + -24.059;
   1:  PR[GP1:91,2] = PR[GP1:90,2] + -41.066;
   1:L PR[91] 10mm/sec CNT100;
   1:  PR[GP1:91,1] = PR[GP1:90,1] + -18.931;
   1:  PR[GP1:91,2] = PR[GP1:90,2] + -42.025;
   1:L PR[91] 10mm/sec CNT100;
   1:  PR[GP1:91,1] = PR[GP1:90,1] + -9.147;
   1:  PR[GP1:91,2] = PR[GP1:90,2] + -43.099;
   1:L PR[91] 10mm/sec CNT100;
   1:  PR[GP1:91,1] = PR[GP1:90,1] + -3.790;
   1:  PR[GP1:91,2] = PR[GP1:90,2] + -42.201;
   1:L PR[91] 10mm/sec CNT100;
   1:  PR[GP1:91,1] = PR[GP1:90,1] + -0.261;
   1:  PR[GP1:91,2] = PR[GP1:90,2] + -41.442;
   1:L PR[91] 10mm/sec CNT100;
   1:  PR[GP1:91,1] = PR[GP1:90,1] + 2.830;
   1:  PR[GP1:91,2] = PR[GP1:90,2] + -42.288;
   1:  PR[GP1:91,3] = PR[GP1:90,3] + 100.345;
   1:L PR[91] 10mm/sec CNT100;
   1:  PR[GP1:91,1] = PR[GP1:90,1] + 8.428;
   1:  PR[GP1:91,2] = PR[GP1:90,2] + -43.228;
   1:L PR[91] 10mm/sec CNT100;
   1:  PR[GP1:91,1] = PR[GP1:90,1] + 18.002;
   1:  PR[GP1:91,2] = PR[GP1:90,2] + -42.176;
   1:L PR[91] 10mm/sec CNT100;
   1:  PR[GP1:91,1] = PR[GP1:90,1] + 23.405;
   1:  PR[GP1:91,2] = PR[GP1:90,2] + -41.166;
   1:L PR[91] 10mm/sec CNT100;
   1:  PR[GP1:91,1] = PR[GP1:90,1] + 32.431;
   1:  PR[GP1:91,2] = PR[GP1:90,2] + -37.046;
   1:L PR[91] 10mm/sec CNT100;
   1:  PR[GP1:91,1] = PR[GP1:90,1] + 36.654;
   1:  PR[GP1:91,2] = PR[GP1:90,2] + -34.431;
   1:L PR[91] 10mm/sec CNT100;
   1:  PR[GP1:91,1] = PR[GP1:90,1] + 44.080;
   1:  PR[GP1:91,2] = PR[GP1:90,2] + -27.527;
   1:L PR[91] 10mm/sec CNT100;
   1:  PR[GP1:91,1] = PR[GP1:90,1] + 46.229;
   1:  PR[GP1:91,2] = PR[GP1:90,2] + -24.939;
   1:L PR[91] 10mm/sec CNT100;
   1:  PR[GP1:91,1] = PR[GP1:90,1] + 51.164;
   1:  PR[GP1:91,2] = PR[GP1:90,2] + -15.860;
   1:L PR[91] 10mm/sec CNT100;
   1:  PR[GP1:91,1] = PR[GP1:90,1] + 52.427;
   1:  PR[GP1:91,2] = PR[GP1:90,2] + -12.998;
   1:L PR[91] 10mm/sec CNT100;
   1:  PR[GP1:91,1] = PR[GP1:90,1] + 54.145;
   1:  PR[GP1:91,2] = PR[GP1:90,2] + -2.775;
   1:L PR[91] 10mm/sec CNT100;
   1:  PR[GP1:91,1] = PR[GP1:90,1] + 54.148;
   1:  PR[GP1:91,2] = PR[GP1:90,2] + -2.524;
   1:L PR[91] 10mm/sec CNT100;
   1:  PR[GP1:91,1] = PR[GP1:90,1] + 54.538;
   1:  PR[GP1:91,2] = PR[GP1:90,2] + 0.271;
   1:L PR[91] 10mm/sec CNT100;
   1:  PR[GP1:91,1] = PR[GP1:90,1] + 52.852;
   1:  PR[GP1:91,2] = PR[GP1:90,2] + 10.462;
   1:L PR[91] 10mm/sec CNT100;
   1:  PR[GP1:91,1] = PR[GP1:90,1] + 52.416;
   1:  PR[GP1:91,2] = PR[GP1:90,2] + 13.585;
   1:L PR[91] 10mm/sec CNT100;
   1:  PR[GP1:91,1] = PR[GP1:90,1] + 51.156;
   1:  PR[GP1:91,2] = PR[GP1:90,2] + 16.439;
   1:L PR[91] 10mm/sec CNT100;
   1:  PR[GP1:91,1] = PR[GP1:90,1] + 46.202;
   1:  PR[GP1:91,2] = PR[GP1:90,2] + 25.531;
   1:L PR[91] 10mm/sec CNT100;
   1:  PR[GP1:91,1] = PR[GP1:90,1] + 44.053;
   1:  PR[GP1:91,2] = PR[GP1:90,2] + 28.121;
   1:L PR[91] 10mm/sec CNT100;
   1:  PR[GP1:91,1] = PR[GP1:90,1] + 36.601;
   1:  PR[GP1:91,2] = PR[GP1:90,2] + 35.024;
   1:L PR[91] 10mm/sec CNT100;
   1:  PR[GP1:91,1] = PR[GP1:90,1] + 32.376;
   1:  PR[GP1:91,2] = PR[GP1:90,2] + 37.641;
   1:L PR[91] 10mm/sec CNT100;
   1:  PR[GP1:91,1] = PR[GP1:90,1] + 23.326;
   1:  PR[GP1:91,2] = PR[GP1:90,2] + 41.746;
   1:L PR[91] 10mm/sec CNT100;
   1:  PR[GP1:91,1] = PR[GP1:90,1] + 17.918;
   1:  PR[GP1:91,2] = PR[GP1:90,2] + 42.757;
   1:L PR[91] 10mm/sec CNT100;
   1:  PR[GP1:91,1] = PR[GP1:90,1] + 8.332;
   1:  PR[GP1:91,2] = PR[GP1:90,2] + 43.780;
   1:L PR[91] 10mm/sec CNT100;
   1:  PR[GP1:91,1] = PR[GP1:90,1] + 0.483;
   1:  PR[GP1:91,2] = PR[GP1:90,2] + 42.400;
   1:L PR[91] 10mm/sec CNT100;
   1:  PR[GP1:91,1] = PR[GP1:90,1] + -0.260;
   1:  PR[GP1:91,2] = PR[GP1:90,2] + 42.238;
   1:L PR[91] 10mm/sec CNT100;
   1:  PR[GP1:91,1] = PR[GP1:90,1] + -1.003;
   1:  PR[GP1:91,2] = PR[GP1:90,2] + 42.400;
   1:L PR[91] 10mm/sec CNT100;
   1:  PR[GP1:91,1] = PR[GP1:90,1] + -8.860;
   1:  PR[GP1:91,2] = PR[GP1:90,2] + 43.780;
   1:L PR[91] 10mm/sec CNT100;
   1:  PR[GP1:91,1] = PR[GP1:90,1] + -18.447;
   1:  PR[GP1:91,2] = PR[GP1:90,2] + 42.758;
   1:L PR[91] 10mm/sec CNT100;
   1:  PR[GP1:91,1] = PR[GP1:90,1] + -23.853;
   1:  PR[GP1:91,2] = PR[GP1:90,2] + 41.746;
   1:L PR[91] 10mm/sec CNT100;
   1:  PR[GP1:91,1] = PR[GP1:90,1] + -32.903;
   1:  PR[GP1:91,2] = PR[GP1:90,2] + 37.638;
   1:L PR[91] 10mm/sec CNT100;
   1:  PR[GP1:91,1] = PR[GP1:90,1] + -37.127;
   1:  PR[GP1:91,2] = PR[GP1:90,2] + 35.022;
   1:L PR[91] 10mm/sec CNT100;
   1:  PR[GP1:91,1] = PR[GP1:90,1] + -44.579;
   1:  PR[GP1:91,2] = PR[GP1:90,2] + 28.127;
   1:L PR[91] 10mm/sec CNT100;
   1:  PR[GP1:91,1] = PR[GP1:90,1] + -46.728;
   1:  PR[GP1:91,2] = PR[GP1:90,2] + 25.538;
   1:L PR[91] 10mm/sec CNT100;
   1:  PR[GP1:91,1] = PR[GP1:90,1] + -51.682;
   1:  PR[GP1:91,2] = PR[GP1:90,2] + 16.429;
   1:L PR[91] 10mm/sec CNT100;
   1:  PR[GP1:91,1] = PR[GP1:90,1] + -52.946;
   1:  PR[GP1:91,2] = PR[GP1:90,2] + 13.566;
   1:L PR[91] 10mm/sec CNT100;
   1:  PR[GP1:91,1] = PR[GP1:90,1] + -54.672;
   1:  PR[GP1:91,2] = PR[GP1:90,2] + 3.333;
   1:L PR[91] 10mm/sec CNT100;
   1:  PR[GP1:91,1] = PR[GP1:90,1] + -54.674;
   1:  PR[GP1:91,2] = PR[GP1:90,2] + 3.083;
   1:L PR[91] 10mm/sec CNT100;
   1:  PR[GP1:91,1] = PR[GP1:90,1] + -55.064;
   1:  PR[GP1:91,2] = PR[GP1:90,2] + 0.287;
   1:L PR[91] 10mm/sec CNT100;
   1:  PR[GP1:91,1] = PR[GP1:90,1] + -53.386;
   1:  PR[GP1:91,2] = PR[GP1:90,2] + -9.872;
   1:L PR[91] 10mm/sec CNT100;
   1:  PR[GP1:91,1] = PR[GP1:90,1] + -52.950;
   1:  PR[GP1:91,2] = PR[GP1:90,2] + -12.995;
   1:L PR[91] 10mm/sec CNT100;
   1:  PR[GP1:91,1] = PR[GP1:90,1] + -51.690;
   1:  PR[GP1:91,2] = PR[GP1:90,2] + -15.849;
   1:L PR[91] 10mm/sec CNT100;
   1:  PR[GP1:91,1] = PR[GP1:90,1] + -46.755;
   1:  PR[GP1:91,2] = PR[GP1:90,2] + -24.945;
   1:L PR[91] 10mm/sec CNT100;
   1:  PR[GP1:91,1] = PR[GP1:90,1] + -44.606;
   1:  PR[GP1:91,2] = PR[GP1:90,2] + -27.533;
   1:L PR[91] 10mm/sec CNT100;
   1:  PR[GP1:91,1] = PR[GP1:90,1] + -37.180;
   1:  PR[GP1:91,2] = PR[GP1:90,2] + -34.429;
   1:L PR[91] 10mm/sec CNT100;
   1:  PR[GP1:91,1] = PR[GP1:90,1] + -32.958;
   1:  PR[GP1:91,2] = PR[GP1:90,2] + -37.044;
   1:L PR[91] 10mm/sec CNT100;
   1:  PR[GP1:91,1] = PR[GP1:90,1] + -23.933;
   1:  PR[GP1:91,2] = PR[GP1:90,2] + -41.167;
   1:L PR[91] 10mm/sec CNT100;
   1:  PR[GP1:91,1] = PR[GP1:90,1] + -18.531;
   1:  PR[GP1:91,2] = PR[GP1:90,2] + -42.177;
   1:L PR[91] 10mm/sec CNT100;
   1:  PR[GP1:91,1] = PR[GP1:90,1] + -8.957;
   1:  PR[GP1:91,2] = PR[GP1:90,2] + -43.228;
   1:L PR[91] 10mm/sec CNT100;
   1:  PR[GP1:91,1] = PR[GP1:90,1] + -3.352;
   1:  PR[GP1:91,2] = PR[GP1:90,2] + -42.288;
   1:L PR[91] 10mm/sec CNT100;
   1:  PR[GP1:91,1] = PR[GP1:90,1] + -0.261;
   1:  PR[GP1:91,2] = PR[GP1:90,2] + -41.623;
   1:L PR[91] 10mm/sec CNT100;
   1:  PR[GP1:91,1] = PR[GP1:90,1] + 2.392;
   1:  PR[GP1:91,2] = PR[GP1:90,2] + -42.375;
   1:  PR[GP1:91,3] = PR[GP1:90,3] + 100.955;
   1:L PR[91] 10mm/sec CNT100;
   1:  PR[GP1:91,1] = PR[GP1:90,1] + 8.239;
   1:  PR[GP1:91,2] = PR[GP1:90,2] + -43.356;
   1:L PR[91] 10mm/sec CNT100;
   1:  PR[GP1:91,1] = PR[GP1:90,1] + 17.602;
   1:  PR[GP1:91,2] = PR[GP1:90,2] + -42.328;
   1:L PR[91] 10mm/sec CNT100;
   1:  PR[GP1:91,1] = PR[GP1:90,1] + 23.279;
   1:  PR[GP1:91,2] = PR[GP1:90,2] + -41.267;
   1:L PR[91] 10mm/sec CNT100;
   1:  PR[GP1:91,1] = PR[GP1:90,1] + 32.106;
   1:  PR[GP1:91,2] = PR[GP1:90,2] + -37.237;
   1:L PR[91] 10mm/sec CNT100;
   1:  PR[GP1:91,1] = PR[GP1:90,1] + 36.576;
   1:  PR[GP1:91,2] = PR[GP1:90,2] + -34.469;
   1:L PR[91] 10mm/sec CNT100;
   1:  PR[GP1:91,1] = PR[GP1:90,1] + 43.838;
   1:  PR[GP1:91,2] = PR[GP1:90,2] + -27.718;
   1:L PR[91] 10mm/sec CNT100;
   1:  PR[GP1:91,1] = PR[GP1:90,1] + 46.132;
   1:  PR[GP1:91,2] = PR[GP1:90,2] + -24.955;
   1:L PR[91] 10mm/sec CNT100;
   1:  PR[GP1:91,1] = PR[GP1:90,1] + 50.958;
   1:  PR[GP1:91,2] = PR[GP1:90,2] + -16.076;
   1:L PR[91] 10mm/sec CNT100;
   1:  PR[GP1:91,1] = PR[GP1:90,1] + 52.314;
   1:  PR[GP1:91,2] = PR[GP1:90,2] + -13.003;
   1:L PR[91] 10mm/sec CNT100;
   1:  PR[GP1:91,1] = PR[GP1:90,1] + 53.994;
   1:  PR[GP1:91,2] = PR[GP1:90,2] + -3.006;
   1:L PR[91] 10mm/sec CNT100;
   1:  PR[GP1:91,1] = PR[GP1:90,1] + 53.997;
   1:  PR[GP1:91,2] = PR[GP1:90,2] + -2.761;
   1:L PR[91] 10mm/sec CNT100;
   1:  PR[GP1:91,1] = PR[GP1:90,1] + 54.420;
   1:  PR[GP1:91,2] = PR[GP1:90,2] + 0.271;
   1:L PR[91] 10mm/sec CNT100;
   1:  PR[GP1:91,1] = PR[GP1:90,1] + 52.771;
   1:  PR[GP1:91,2] = PR[GP1:90,2] + 10.238;
   1:L PR[91] 10mm/sec CNT100;
   1:  PR[GP1:91,1] = PR[GP1:90,1] + 52.304;
   1:  PR[GP1:91,2] = PR[GP1:90,2] + 13.589;
   1:L PR[91] 10mm/sec CNT100;
   1:  PR[GP1:91,1] = PR[GP1:90,1] + 50.950;
   1:  PR[GP1:91,2] = PR[GP1:90,2] + 16.655;
   1:L PR[91] 10mm/sec CNT100;
   1:  PR[GP1:91,1] = PR[GP1:90,1] + 46.105;
   1:  PR[GP1:91,2] = PR[GP1:90,2] + 25.547;
   1:L PR[91] 10mm/sec CNT100;
   1:  PR[GP1:91,1] = PR[GP1:90,1] + 43.811;
   1:  PR[GP1:91,2] = PR[GP1:90,2] + 28.310;
   1:L PR[91] 10mm/sec CNT100;
   1:  PR[GP1:91,1] = PR[GP1:90,1] + 36.524;
   1:  PR[GP1:91,2] = PR[GP1:90,2] + 35.061;
   1:L PR[91] 10mm/sec CNT100;
   1:  PR[GP1:91,1] = PR[GP1:90,1] + 32.052;
   1:  PR[GP1:91,2] = PR[GP1:90,2] + 37.831;
   1:L PR[91] 10mm/sec CNT100;
   1:  PR[GP1:91,1] = PR[GP1:90,1] + 23.202;
   1:  PR[GP1:91,2] = PR[GP1:90,2] + 41.846;
   1:L PR[91] 10mm/sec CNT100;
   1:  PR[GP1:91,1] = PR[GP1:90,1] + 17.520;
   1:  PR[GP1:91,2] = PR[GP1:90,2] + 42.908;
   1:L PR[91] 10mm/sec CNT100;
   1:  PR[GP1:91,1] = PR[GP1:90,1] + 8.145;
   1:  PR[GP1:91,2] = PR[GP1:90,2] + 43.909;
   1:L PR[91] 10mm/sec CNT100;
   1:  PR[GP1:91,1] = PR[GP1:90,1] + -0.260;
   1:  PR[GP1:91,2] = PR[GP1:90,2] + 42.427;
   1:L PR[91] 10mm/sec CNT100;
   1:  PR[GP1:91,1] = PR[GP1:90,1] + -8.673;
   1:  PR[GP1:91,2] = PR[GP1:90,2] + 43.909;
   1:L PR[91] 10mm/sec CNT100;
   1:  PR[GP1:91,1] = PR[GP1:90,1] + -18.048;
   1:  PR[GP1:91,2] = PR[GP1:90,2] + 42.909;
   1:L PR[91] 10mm/sec CNT100;
   1:  PR[GP1:91,1] = PR[GP1:90,1] + -23.728;
   1:  PR[GP1:91,2] = PR[GP1:90,2] + 41.846;
   1:L PR[91] 10mm/sec CNT100;
   1:  PR[GP1:91,1] = PR[GP1:90,1] + -32.578;
   1:  PR[GP1:91,2] = PR[GP1:90,2] + 37.829;
   1:L PR[91] 10mm/sec CNT100;
   1:  PR[GP1:91,1] = PR[GP1:90,1] + -37.050;
   1:  PR[GP1:91,2] = PR[GP1:90,2] + 35.059;
   1:L PR[91] 10mm/sec CNT100;
   1:  PR[GP1:91,1] = PR[GP1:90,1] + -44.337;
   1:  PR[GP1:91,2] = PR[GP1:90,2] + 28.317;
   1:L PR[91] 10mm/sec CNT100;
   1:  PR[GP1:91,1] = PR[GP1:90,1] + -46.631;
   1:  PR[GP1:91,2] = PR[GP1:90,2] + 25.553;
   1:L PR[91] 10mm/sec CNT100;
   1:  PR[GP1:91,1] = PR[GP1:90,1] + -51.476;
   1:  PR[GP1:91,2] = PR[GP1:90,2] + 16.645;
   1:L PR[91] 10mm/sec CNT100;
   1:  PR[GP1:91,1] = PR[GP1:90,1] + -52.833;
   1:  PR[GP1:91,2] = PR[GP1:90,2] + 13.571;
   1:L PR[91] 10mm/sec CNT100;
   1:  PR[GP1:91,1] = PR[GP1:90,1] + -54.521;
   1:  PR[GP1:91,2] = PR[GP1:90,2] + 3.564;
   1:L PR[91] 10mm/sec CNT100;
   1:  PR[GP1:91,1] = PR[GP1:90,1] + -54.523;
   1:  PR[GP1:91,2] = PR[GP1:90,2] + 3.319;
   1:L PR[91] 10mm/sec CNT100;
   1:  PR[GP1:91,1] = PR[GP1:90,1] + -54.946;
